LIN {X 0,Y 221.145,Z 638.431,A -85,B 0,C 180,E1 -21909.464,E2 -21909.464} C_VEL
LIN {X 0,Y 225.673,Z 625.218,A -85,B 0,C 180,E1 -21911.415,E2 -21911.415} C_VEL
LIN {X 0,Y 229.459,Z 612.073,A -85,B 0,C 180,E1 -21912.96,E2 -21912.96} C_VEL
LIN {X 0,Y 232.879,Z 597.827,A -85,B 0,C 180,E1 -21914.257,E2 -21914.257} C_VEL
LIN {X 0,Y 235.879,Z 582.403,A -85,B 0,C 180,E1 -21915.269,E2 -21915.269} C_VEL
LIN {X 0,Y 237.953,Z 566.942,A -85,B 0,C 180,E1 -21915.972,E2 -21915.972} C_VEL
LIN {X 0,Y 240.422,Z 531.68,A -85,B 0,C 180,E1 -21916.953,E2 -21916.953} C_VEL
LIN {X 0,Y 244.484,Z 467.241,A -85,B 0,C 180,E1 -21918.681,E2 -21918.681} C_VEL
LIN {X 0,Y 239.527,Z 455.727,A -85,B 0,C 180,E1 -21920.57,E2 -21920.57} C_VEL
LIN {X 0,Y 234.309,Z 445.003,A -85,B 0,C 180,E1 -21922.666,E2 -21922.666} C_VEL
LIN {X 0,Y 227.784,Z 433.109,A -85,B 0,C 180,E1 -21925.503,E2 -21925.503} C_VEL
LIN {X 0,Y 221.655,Z 423.149,A -85,B 0,C 180,E1 -21928.464,E2 -21928.464} C_VEL
LIN {X 0,Y 217.57,Z 417.19,A -85,B 0,C 180,E1 -21930.641,E2 -21930.641} C_VEL
LIN {X 0,Y 213.973,Z 412.042,A -85,B 0,C 180,E1 -21932.756,E2 -21932.756} C_VEL
LIN {X 0,Y 209.301,Z 405.782,A -85,B 0,C 180,E1 -21935.843,E2 -21935.843} C_VEL
LIN {X 0,Y 204.867,Z 400.056,A -85,B 0,C 180,E1 -21939.298,E2 -21939.298} C_VEL
LIN {X 0,Y 200.557,Z 394.827,A -85,B 0,C 180,E1 -21943.458,E2 -21943.458} C_VEL
LIN {X 0,Y 198.701,Z 391.203,A -85,B 0,C 180,E1 -21947.747,E2 -21947.747} C_VEL
LIN {X 0,Y 197.369,Z 389.174,A -85,B 0,C 180,E1 -21951.811,E2 -21951.811} C_VEL
LIN {X 0,Y 196.672,Z 386.877,A -85,B 0,C 180,E1 -21957.952,E2 -21957.952} C_VEL
LIN {X 0,Y 196.702,Z 386.437,A -85,B 0,C 180,E1 -21960,E2 -21960} C_VEL
LIN {X 0,Y 196.636,Z 386.629,A -85,B 0,C 180,E1 -21962.048,E2 -21962.048} C_VEL
LIN {X 0,Y 197.132,Z 388.567,A -85,B 0,C 180,E1 -21968.198,E2 -21968.198} C_VEL
LIN {X 0,Y 199.318,Z 391.66,A -85,B 0,C 180,E1 -21974.289,E2 -21974.289} C_VEL
LIN {X 0,Y 199.881,Z 392.9,A -85,B 0,C 180,E1 -21975.695,E2 -21975.695} C_VEL
LIN {X 0,Y 200.923,Z 394.996,A -85,B 0,C 180,E1 -21977.237,E2 -21977.237} C_VEL
LIN {X 0,Y 202.106,Z 398.063,A -85,B 0,C 180,E1 -21978.639,E2 -21978.639} C_VEL
LIN {X 0,Y 205.482,Z 407.511,A -85,B 0,C 180,E1 -21982.147,E2 -21982.147} C_VEL
LIN {X 0,Y 206.581,Z 409.464,A -85,B 0,C 180,E1 -21983.069,E2 -21983.069} C_VEL
LIN {X 0,Y 210.001,Z 413.782,A -85,B 0,C 180,E1 -21985.523,E2 -21985.523} C_VEL
LIN {X 0,Y 213.678,Z 418.756,A -85,B 0,C 180,E1 -21987.882,E2 -21987.882} C_VEL
LIN {X 0,Y 217.594,Z 424.126,A -85,B 0,C 180,E1 -21990.134,E2 -21990.134} C_VEL
LIN {X 0,Y 222.494,Z 431.302,A -85,B 0,C 180,E1 -21992.678,E2 -21992.678} C_VEL
LIN {X 0,Y 228.634,Z 440.96,A -85,B 0,C 180,E1 -21995.532,E2 -21995.532} C_VEL
LIN {X 0,Y 234.218,Z 450.7,A -85,B 0,C 180,E1 -21997.893,E2 -21997.893} C_VEL
LIN {X 0,Y 239.469,Z 465.456,A -85,B 0,C 180,E1 -22000.165,E2 -22000.165} C_VEL
LIN {X 0,Y 232.939,Z 563.19,A -85,B 0,C 180,E1 -22002.817,E2 -22002.817} C_VEL
LIN {X 0,Y 231.11,Z 578.287,A -85,B 0,C 180,E1 -22003.445,E2 -22003.445} C_VEL
LIN {X 0,Y 228.399,Z 593.01,A -85,B 0,C 180,E1 -22004.323,E2 -22004.323} C_VEL
LIN {X 0,Y 225.305,Z 606.361,A -85,B 0,C 180,E1 -22005.425,E2 -22005.425} C_VEL
LIN {X 0,Y 221.488,Z 620.138,A -85,B 0,C 180,E1 -22006.924,E2 -22006.924} C_VEL
LIN {X 0,Y 217.136,Z 633.278,A -85,B 0,C 180,E1 -22008.74,E2 -22008.74} C_VEL
LIN {X 0,Y 212.533,Z 645.127,A -85,B 0,C 180,E1 -22010.771,E2 -22010.771} C_VEL
LIN {X 0,Y 207.922,Z 656.085,A -85,B 0,C 180,E1 -22013.133,E2 -22013.133} C_VEL
LIN {X 0,Y 203.231,Z 666.179,A -85,B 0,C 180,E1 -22015.81,E2 -22015.81} C_VEL
LIN {X 0,Y 199.177,Z 674.689,A -85,B 0,C 180,E1 -22018.637,E2 -22018.637} C_VEL
LIN {X 0,Y 194.766,Z 683.074,A -85,B 0,C 180,E1 -22022.025,E2 -22022.025} C_VEL
LIN {X 0,Y 190.712,Z 690.93,A -85,B 0,C 180,E1 -22026.086,E2 -22026.086} C_VEL
LIN {X 0,Y 187.54,Z 697.179,A -85,B 0,C 180,E1 -22030.289,E2 -22030.289} C_VEL
LIN {X 0,Y 185.261,Z 701.999,A -85,B 0,C 180,E1 -22034.601,E2 -22034.601} C_VEL
LIN {X 0,Y 183.848,Z 705.52,A -85,B 0,C 180,E1 -22038.981,E2 -22038.981} C_VEL
LIN {X 0,Y 183.137,Z 707.835,A -85,B 0,C 180,E1 -22043.389,E2 -22043.389} C_VEL
LIN {X 0,Y 183.02,Z 708.996,A -85,B 0,C 180,E1 -22047.8,E2 -22047.8} C_VEL
LIN {X 0,Y 183.031,Z 709.146,A -85,B 0,C 180,E1 -22050,E2 -22050} C_VEL
LIN {X 0,Y 183.073,Z 708.547,A -85,B 0,C 180,E1 -22054.404,E2 -22054.404} C_VEL
LIN {X 0,Y 183.407,Z 706.799,A -85,B 0,C 180,E1 -22058.817,E2 -22058.817} C_VEL
LIN {X 0,Y 184.445,Z 703.868,A -85,B 0,C 180,E1 -22063.216,E2 -22063.216} C_VEL
LIN {X 0,Y 186.337,Z 699.686,A -85,B 0,C 180,E1 -22067.562,E2 -22067.562} C_VEL
LIN {X 0,Y 188.987,Z 694.152,A -85,B 0,C 180,E1 -22071.832,E2 -22071.832} C_VEL
LIN {X 0,Y 191.461,Z 689.781,A -85,B 0,C 180,E1 -22074.68,E2 -22074.68} C_VEL
LIN {X 0,Y 197.957,Z 686.616,A -85,B 0,C 180,E1 -22079.804,E2 -22079.804} C_VEL
LIN {X 0,Y 204.195,Z 683.167,A -85,B 0,C 180,E1 -22083.415,E2 -22083.415} C_VEL
LIN {X 0,Y 211.419,Z 678.76,A -85,B 0,C 180,E1 -22086.753,E2 -22086.753} C_VEL
LIN {X 0,Y 221.903,Z 671.855,A -85,B 0,C 180,E1 -22090.487,E2 -22090.487} C_VEL
LIN {X 0,Y 231.146,Z 665.173,A -85,B 0,C 180,E1 -22093.166,E2 -22093.166} C_VEL
LIN {X 0,Y 242.53,Z 656.247,A -85,B 0,C 180,E1 -22095.824,E2 -22095.824} C_VEL
LIN {X 0,Y 246.76,Z 652.737,A -85,B 0,C 180,E1 -22096.694,E2 -22096.694} C_VEL
LIN {X 0,Y 248.311,Z 651.353,A -85,B 0,C 180,E1 -22097.213,E2 -22097.213} C_VEL
LIN {X 0,Y 238.076,Z 658.959,A -85,B 0,C 180,E1 -22099.501,E2 -22099.501} C_VEL
LIN {X 0,Y 228.584,Z 665.287,A -85,B 0,C 180,E1 -22102.054,E2 -22102.054} C_VEL
LIN {X 0,Y 219.85,Z 670.441,A -85,B 0,C 180,E1 -22104.872,E2 -22104.872} C_VEL
LIN {X 0,Y 211.838,Z 674.517,A -85,B 0,C 180,E1 -22107.939,E2 -22107.939} C_VEL
LIN {X 0,Y 204.688,Z 677.495,A -85,B 0,C 180,E1 -22111.27,E2 -22111.27} C_VEL
LIN {X 0,Y 198.621,Z 679.336,A -85,B 0,C 180,E1 -22114.874,E2 -22114.874} C_VEL
LIN {X 0,Y 193.513,Z 680.122,A -85,B 0,C 180,E1 -22118.705,E2 -22118.705} C_VEL
LIN {X 0,Y 189.625,Z 679.823,A -85,B 0,C 180,E1 -22122.753,E2 -22122.753} C_VEL
LIN {X 0,Y 186.665,Z 678.421,A -85,B 0,C 180,E1 -22126.944,E2 -22126.944} C_VEL
LIN {X 0,Y 184.683,Z 675.852,A -85,B 0,C 180,E1 -22131.245,E2 -22131.245} C_VEL
LIN {X 0,Y 183.798,Z 672.043,A -85,B 0,C 180,E1 -22135.614,E2 -22135.614} C_VEL
LIN {X 0,Y 183.535,Z 668.25,A -85,B 0,C 180,E1 -22138.903,E2 -22138.903} C_VEL
LIN {X 0,Y 183.475,Z 663.633,A -85,B 0,C 180,E1 -22142.195,E2 -22142.195} C_VEL
LIN {X 0,Y 183.761,Z 655.877,A -85,B 0,C 180,E1 -22146.589,E2 -22146.589} C_VEL
LIN {X 0,Y 184.363,Z 647.395,A -85,B 0,C 180,E1 -22150.432,E2 -22150.432} C_VEL
LIN {X 0,Y 185.232,Z 638.646,A -85,B 0,C 180,E1 -22153.718,E2 -22153.718} C_VEL
LIN {X 0,Y 186.582,Z 628.253,A -85,B 0,C 180,E1 -22156.973,E2 -22156.973} C_VEL
LIN {X 0,Y 188.232,Z 616.073,A -85,B 0,C 180,E1 -22160.138,E2 -22160.138} C_VEL
LIN {X 0,Y 190.004,Z 603.327,A -85,B 0,C 180,E1 -22162.853,E2 -22162.853} C_VEL
LIN {X 0,Y 191.936,Z 589.886,A -85,B 0,C 180,E1 -22165.193,E2 -22165.193} C_VEL
LIN {X 0,Y 193.983,Z 574.43,A -85,B 0,C 180,E1 -22167.366,E2 -22167.366} C_VEL
LIN {X 0,Y 194.89,Z 567.266,A -85,B 0,C 180,E1 -22168.396,E2 -22168.396} C_VEL
LIN {X 0,Y 195.611,Z 564.799,A -85,B 0,C 180,E1 -22169.015,E2 -22169.015} C_VEL
LIN {X 0,Y 197.306,Z 562.863,A -85,B 0,C 180,E1 -22169.839,E2 -22169.839} C_VEL
LIN {X 0,Y 199.619,Z 558.803,A -85,B 0,C 180,E1 -22170.624,E2 -22170.624} C_VEL
LIN {X 0,Y 202.727,Z 550.321,A -85,B 0,C 180,E1 -22171.506,E2 -22171.506} C_VEL
LIN {X 0,Y 207.709,Z 533.515,A -85,B 0,C 180,E1 -22172.634,E2 -22172.634} C_VEL
LIN {X 0,Y 209.994,Z 530.321,A -85,B 0,C 180,E1 -22173.397,E2 -22173.397} C_VEL
LIN {X 0,Y 212.304,Z 525.327,A -85,B 0,C 180,E1 -22174.034,E2 -22174.034} C_VEL
LIN {X 0,Y 216.015,Z 514.502,A -85,B 0,C 180,E1 -22174.848,E2 -22174.848} C_VEL
LIN {X 0,Y 221.035,Z 497.363,A -85,B 0,C 180,E1 -22175.746,E2 -22175.746} C_VEL
LIN {X 0,Y 223.977,Z 492.781,A -85,B 0,C 180,E1 -22176.534,E2 -22176.534} C_VEL
LIN {X 0,Y 227.199,Z 485.435,A -85,B 0,C 180,E1 -22177.239,E2 -22177.239} C_VEL
LIN {X 0,Y 230.92,Z 474.319,A -85,B 0,C 180,E1 -22177.885,E2 -22177.885} C_VEL
LIN {X 0,Y 234.212,Z 463.118,A -85,B 0,C 180,E1 -22178.366,E2 -22178.366} C_VEL
LIN {X 0,Y 235.788,Z 461.138,A -85,B 0,C 180,E1 -22178.751,E2 -22178.751} C_VEL
LIN {X 0,Y 238.047,Z 465.902,A -85,B 0,C 180,E1 -22179.642,E2 -22179.642} C_VEL
LIN {X 0,Y 239.544,Z 469.549,A -85,B 0,C 180,E1 -22180.237,E2 -22180.237} C_VEL
LIN {X 0,Y 234.668,Z 543.882,A -85,B 0,C 180,E1 -22182.243,E2 -22182.243} C_VEL
LIN {X 0,Y 232.919,Z 566.712,A -85,B 0,C 180,E1 -22182.89,E2 -22182.89} C_VEL
LIN {X 0,Y 230.795,Z 582.245,A -85,B 0,C 180,E1 -22183.6,E2 -22183.6} C_VEL
LIN {X 0,Y 227.711,Z 597.718,A -85,B 0,C 180,E1 -22184.619,E2 -22184.619} C_VEL
LIN {X 0,Y 224.425,Z 611.093,A -85,B 0,C 180,E1 -22185.831,E2 -22185.831} C_VEL
LIN {X 0,Y 220.636,Z 624.081,A -85,B 0,C 180,E1 -22187.36,E2 -22187.36} C_VEL
LIN {X 0,Y 215.819,Z 637.746,A -85,B 0,C 180,E1 -22189.361,E2 -22189.361} C_VEL
LIN {X 0,Y 210.958,Z 649.959,A -85,B 0,C 180,E1 -22191.648,E2 -22191.648} C_VEL
LIN {X 0,Y 205.603,Z 661.938,A -85,B 0,C 180,E1 -22194.472,E2 -22194.472} C_VEL
LIN {X 0,Y 200.757,Z 672.218,A -85,B 0,C 180,E1 -22197.57,E2 -22197.57} C_VEL
LIN {X 0,Y 196.656,Z 680.261,A -85,B 0,C 180,E1 -22200.568,E2 -22200.568} C_VEL
LIN {X 0,Y 192.717,Z 687.801,A -85,B 0,C 180,E1 -22204.048,E2 -22204.048} C_VEL
LIN {X 0,Y 189.086,Z 694.833,A -85,B 0,C 180,E1 -22208.18,E2 -22208.18} C_VEL
LIN {X 0,Y 186.404,Z 700.363,A -85,B 0,C 180,E1 -22212.445,E2 -22212.445} C_VEL
LIN {X 0,Y 184.461,Z 704.547,A -85,B 0,C 180,E1 -22216.785,E2 -22216.785} C_VEL
LIN {X 0,Y 183.41,Z 707.485,A -85,B 0,C 180,E1 -22221.183,E2 -22221.183} C_VEL
LIN {X 0,Y 183.015,Z 709.245,A -85,B 0,C 180,E1 -22225.595,E2 -22225.595} C_VEL
LIN {X 0,Y 183.028,Z 709.852,A -85,B 0,C 180,E1 -22230,E2 -22230} C_VEL
LIN {X 0,Y 183.015,Z 709.275,A -85,B 0,C 180,E1 -22234.405,E2 -22234.405} C_VEL
LIN {X 0,Y 183.409,Z 707.556,A -85,B 0,C 180,E1 -22238.816,E2 -22238.816} C_VEL
LIN {X 0,Y 184.449,Z 704.665,A -85,B 0,C 180,E1 -22243.215,E2 -22243.215} C_VEL
LIN {X 0,Y 186.36,Z 700.533,A -85,B 0,C 180,E1 -22247.559,E2 -22247.559} C_VEL
LIN {X 0,Y 188.988,Z 695.048,A -85,B 0,C 180,E1 -22251.831,E2 -22251.831} C_VEL
LIN {X 0,Y 192.642,Z 688.063,A -85,B 0,C 180,E1 -22255.962,E2 -22255.962} C_VEL
LIN {X 0,Y 196.578,Z 680.583,A -85,B 0,C 180,E1 -22259.445,E2 -22259.445} C_VEL
LIN {X 0,Y 200.549,Z 672.82,A -85,B 0,C 180,E1 -22262.359,E2 -22262.359} C_VEL
LIN {X 0,Y 204.713,Z 663.972,A -85,B 0,C 180,E1 -22265.102,E2 -22265.102} C_VEL
LIN {X 0,Y 209.575,Z 653.397,A -85,B 0,C 180,E1 -22267.734,E2 -22267.734} C_VEL
LIN {X 0,Y 214.332,Z 641.871,A -85,B 0,C 180,E1 -22270.054,E2 -22270.054} C_VEL
LIN {X 0,Y 218.996,Z 629.303,A -85,B 0,C 180,E1 -22272.06,E2 -22272.06} C_VEL
LIN {X 0,Y 223.324,Z 615.487,A -85,B 0,C 180,E1 -22273.815,E2 -22273.815} C_VEL
LIN {X 0,Y 227.053,Z 601.067,A -85,B 0,C 180,E1 -22275.234,E2 -22275.234} C_VEL
LIN {X 0,Y 230.223,Z 586.022,A -85,B 0,C 180,E1 -22276.311,E2 -22276.311} C_VEL
LIN {X 0,Y 232.53,Z 571.213,A -85,B 0,C 180,E1 -22277.053,E2 -22277.053} C_VEL
LIN {X 0,Y 234.057,Z 554.756,A -85,B 0,C 180,E1 -22277.601,E2 -22277.601} C_VEL
LIN {X 0,Y 239.721,Z 469.822,A -85,B 0,C 180,E1 -22279.869,E2 -22279.869} C_VEL
LIN {X 0,Y 235.05,Z 458.909,A -85,B 0,C 180,E1 -22281.755,E2 -22281.755} C_VEL
LIN {X 0,Y 230.72,Z 449.849,A -85,B 0,C 180,E1 -22283.595,E2 -22283.595} C_VEL
LIN {X 0,Y 224.812,Z 438.744,A -85,B 0,C 180,E1 -22286.296,E2 -22286.296} C_VEL
LIN {X 0,Y 219.094,Z 429.197,A -85,B 0,C 180,E1 -22289.187,E2 -22289.187} C_VEL
LIN {X 0,Y 215.01,Z 423.058,A -85,B 0,C 180,E1 -22291.467,E2 -22291.467} C_VEL
LIN {X 0,Y 211.775,Z 418.254,A -85,B 0,C 180,E1 -22293.463,E2 -22293.463} C_VEL
LIN {X 0,Y 207.224,Z 411.967,A -85,B 0,C 180,E1 -22296.615,E2 -22296.615} C_VEL
LIN {X 0,Y 203.203,Z 406.629,A -85,B 0,C 180,E1 -22299.897,E2 -22299.897} C_VEL
LIN {X 0,Y 199.028,Z 401.431,A -85,B 0,C 180,E1 -22304.107,E2 -22304.107} C_VEL
LIN {X 0,Y 195.577,Z 397.2,A -85,B 0,C 180,E1 -22308.863,E2 -22308.863} C_VEL
LIN {X 0,Y 193.057,Z 394.152,A -85,B 0,C 180,E1 -22314.778,E2 -22314.778} C_VEL
LIN {X 0,Y 192.936,Z 392.985,A -85,B 0,C 180,E1 -22317.912,E2 -22317.912} C_VEL
LIN {X 0,Y 193.023,Z 392.513,A -85,B 0,C 180,E1 -22320,E2 -22320} C_VEL
LIN {X 0,Y 192.98,Z 392.732,A -85,B 0,C 180,E1 -22322.087,E2 -22322.087} C_VEL
LIN {X 0,Y 193.62,Z 394.522,A -85,B 0,C 180,E1 -22327.299,E2 -22327.299} C_VEL
LIN {X 0,Y 197.673,Z 398.839,A -85,B 0,C 180,E1 -22334.411,E2 -22334.411} C_VEL
LIN {X 0,Y 202.371,Z 404.31,A -85,B 0,C 180,E1 -22339.527,E2 -22339.527} C_VEL
LIN {X 0,Y 206.581,Z 409.464,A -85,B 0,C 180,E1 -22343.069,E2 -22343.069} C_VEL
LIN {X 0,Y 208.227,Z 412.598,A -85,B 0,C 180,E1 -22344.376,E2 -22344.376} C_VEL
LIN {X 0,Y 213.629,Z 427.51,A -85,B 0,C 180,E1 -22348.471,E2 -22348.471} C_VEL
LIN {X 0,Y 214.927,Z 429.826,A -85,B 0,C 180,E1 -22349.263,E2 -22349.263} C_VEL
LIN {X 0,Y 219.451,Z 436.637,A -85,B 0,C 180,E1 -22351.737,E2 -22351.737} C_VEL
LIN {X 0,Y 225.346,Z 446.156,A -85,B 0,C 180,E1 -22354.625,E2 -22354.625} C_VEL
LIN {X 0,Y 230.661,Z 455.683,A -85,B 0,C 180,E1 -22356.99,E2 -22356.99} C_VEL
LIN {X 0,Y 234.817,Z 467.821,A -85,B 0,C 180,E1 -22358.907,E2 -22358.907} C_VEL
LIN {X 0,Y 228.174,Z 563.309,A -85,B 0,C 180,E1 -22361.509,E2 -22361.509} C_VEL
LIN {X 0,Y 226.298,Z 578.362,A -85,B 0,C 180,E1 -22362.143,E2 -22362.143} C_VEL
LIN {X 0,Y 223.509,Z 593.064,A -85,B 0,C 180,E1 -22363.024,E2 -22363.024} C_VEL
LIN {X 0,Y 220.303,Z 606.404,A -85,B 0,C 180,E1 -22364.129,E2 -22364.129} C_VEL
LIN {X 0,Y 216.479,Z 619.733,A -85,B 0,C 180,E1 -22365.58,E2 -22365.58} C_VEL
LIN {X 0,Y 211.849,Z 633.307,A -85,B 0,C 180,E1 -22367.474,E2 -22367.474} C_VEL
LIN {X 0,Y 207.08,Z 645.152,A -85,B 0,C 180,E1 -22369.528,E2 -22369.528} C_VEL
LIN {X 0,Y 202.257,Z 656.108,A -85,B 0,C 180,E1 -22371.919,E2 -22371.919} C_VEL
LIN {X 0,Y 197.372,Z 666.2,A -85,B 0,C 180,E1 -22374.646,E2 -22374.646} C_VEL
LIN {X 0,Y 194.301,Z 672.289,A -85,B 0,C 180,E1 -22376.646,E2 -22376.646} C_VEL
LIN {X 0,Y 189.721,Z 680.876,A -85,B 0,C 180,E1 -22379.994,E2 -22379.994} C_VEL
LIN {X 0,Y 185.167,Z 689.149,A -85,B 0,C 180,E1 -22384.121,E2 -22384.121} C_VEL
LIN {X 0,Y 181.661,Z 695.501,A -85,B 0,C 180,E1 -22388.202,E2 -22388.202} C_VEL
LIN {X 0,Y 178.942,Z 700.957,A -85,B 0,C 180,E1 -22392.869,E2 -22392.869} C_VEL
LIN {X 0,Y 177.481,Z 703.93,A -85,B 0,C 180,E1 -22396.256,E2 -22396.256} C_VEL
LIN {X 0,Y 176.353,Z 706.839,A -85,B 0,C 180,E1 -22400.828,E2 -22400.828} C_VEL
LIN {X 0,Y 175.969,Z 708.572,A -85,B 0,C 180,E1 -22405.419,E2 -22405.419} C_VEL
LIN {X 0,Y 175.946,Z 709.16,A -85,B 0,C 180,E1 -22410,E2 -22410} C_VEL
LIN {X 0,Y 175.97,Z 708.561,A -85,B 0,C 180,E1 -22414.582,E2 -22414.582} C_VEL
LIN {X 0,Y 176.353,Z 706.812,A -85,B 0,C 180,E1 -22419.173,E2 -22419.173} C_VEL
LIN {X 0,Y 177.483,Z 703.881,A -85,B 0,C 180,E1 -22423.745,E2 -22423.745} C_VEL
LIN {X 0,Y 179.514,Z 699.7,A -85,B 0,C 180,E1 -22428.253,E2 -22428.253} C_VEL
LIN {X 0,Y 182.354,Z 694.166,A -85,B 0,C 180,E1 -22432.669,E2 -22432.669} C_VEL
LIN {X 0,Y 184.976,Z 689.731,A -85,B 0,C 180,E1 -22435.607,E2 -22435.607} C_VEL
LIN {X 0,Y 191.816,Z 686.999,A -85,B 0,C 180,E1 -22440.861,E2 -22440.861} C_VEL
LIN {X 0,Y 198.348,Z 683.928,A -85,B 0,C 180,E1 -22444.536,E2 -22444.536} C_VEL
LIN {X 0,Y 205.866,Z 679.965,A -85,B 0,C 180,E1 -22447.916,E2 -22447.916} C_VEL
LIN {X 0,Y 216.709,Z 673.66,A -85,B 0,C 180,E1 -22451.669,E2 -22451.669} C_VEL
LIN {X 0,Y 228.77,Z 665.813,A -85,B 0,C 180,E1 -22454.958,E2 -22454.958} C_VEL
LIN {X 0,Y 237.539,Z 659.537,A -85,B 0,C 180,E1 -22456.909,E2 -22456.909} C_VEL
LIN {X 0,Y 238.3,Z 658.944,A -85,B 0,C 180,E1 -22457.288,E2 -22457.288} C_VEL
LIN {X 0,Y 228.177,Z 665.279,A -85,B 0,C 180,E1 -22459.698,E2 -22459.698} C_VEL
LIN {X 0,Y 218.763,Z 670.502,A -85,B 0,C 180,E1 -22462.382,E2 -22462.382} C_VEL
LIN {X 0,Y 210.096,Z 674.614,A -85,B 0,C 180,E1 -22465.343,E2 -22465.343} C_VEL
LIN {X 0,Y 202.137,Z 677.686,A -85,B 0,C 180,E1 -22468.566,E2 -22468.566} C_VEL
LIN {X 0,Y 195.325,Z 679.663,A -85,B 0,C 180,E1 -22472.112,E2 -22472.112} C_VEL
LIN {X 0,Y 189.461,Z 680.637,A -85,B 0,C 180,E1 -22475.918,E2 -22475.918} C_VEL
LIN {X 0,Y 184.785,Z 680.556,A -85,B 0,C 180,E1 -22479.983,E2 -22479.983} C_VEL
LIN {X 0,Y 181.163,Z 679.359,A -85,B 0,C 180,E1 -22484.243,E2 -22484.243} C_VEL
LIN {X 0,Y 178.611,Z 677.044,A -85,B 0,C 180,E1 -22488.654,E2 -22488.654} C_VEL
LIN {X 0,Y 177.05,Z 673.543,A -85,B 0,C 180,E1 -22493.161,E2 -22493.161} C_VEL
LIN {X 0,Y 176.576,Z 668.761,A -85,B 0,C 180,E1 -22497.719,E2 -22497.719} C_VEL
LIN {X 0,Y 176.452,Z 664.212,A -85,B 0,C 180,E1 -22501.141,E2 -22501.141} C_VEL
LIN {X 0,Y 176.59,Z 657.403,A -85,B 0,C 180,E1 -22505.267,E2 -22505.267} C_VEL
LIN {X 0,Y 177.114,Z 649.531,A -85,B 0,C 180,E1 -22509.133,E2 -22509.133} C_VEL
LIN {X 0,Y 178.03,Z 639.591,A -85,B 0,C 180,E1 -22513.12,E2 -22513.12} C_VEL
LIN {X 0,Y 179.321,Z 629.357,A -85,B 0,C 180,E1 -22516.508,E2 -22516.508} C_VEL
LIN {X 0,Y 180.953,Z 617.112,A -85,B 0,C 180,E1 -22519.867,E2 -22519.867} C_VEL
LIN {X 0,Y 182.858,Z 603.514,A -85,B 0,C 180,E1 -22522.902,E2 -22522.902} C_VEL
LIN {X 0,Y 185.215,Z 587.713,A -85,B 0,C 180,E1 -22525.873,E2 -22525.873} C_VEL
LIN {X 0,Y 185.81,Z 585.76,A -85,B 0,C 180,E1 -22526.538,E2 -22526.538} C_VEL
LIN {X 0,Y 186.309,Z 585.526,A -85,B 0,C 180,E1 -22526.915,E2 -22526.915} C_VEL
LIN {X 0,Y 188.814,Z 583.488,A -85,B 0,C 180,E1 -22528.03,E2 -22528.03} C_VEL
LIN {X 0,Y 191.85,Z 579.114,A -85,B 0,C 180,E1 -22528.985,E2 -22528.985} C_VEL
LIN {X 0,Y 196.432,Z 570.642,A -85,B 0,C 180,E1 -22530.201,E2 -22530.201} C_VEL
LIN {X 0,Y 198.964,Z 568.102,A -85,B 0,C 180,E1 -22531.141,E2 -22531.141} C_VEL
LIN {X 0,Y 201.887,Z 563.31,A -85,B 0,C 180,E1 -22532.06,E2 -22532.06} C_VEL
LIN {X 0,Y 205.229,Z 555.197,A -85,B 0,C 180,E1 -22532.932,E2 -22532.932} C_VEL
LIN {X 0,Y 209.055,Z 542.703,A -85,B 0,C 180,E1 -22533.763,E2 -22533.763} C_VEL
LIN {X 0,Y 210.533,Z 537.912,A -85,B 0,C 180,E1 -22534.073,E2 -22534.073} C_VEL
LIN {X 0,Y 213.531,Z 533.131,A -85,B 0,C 180,E1 -22534.967,E2 -22534.967} C_VEL
LIN {X 0,Y 216.361,Z 526.461,A -85,B 0,C 180,E1 -22535.651,E2 -22535.651} C_VEL
LIN {X 0,Y 220.395,Z 514.599,A -85,B 0,C 180,E1 -22536.45,E2 -22536.45} C_VEL
LIN {X 0,Y 224.382,Z 501.19,A -85,B 0,C 180,E1 -22537.111,E2 -22537.111} C_VEL
LIN {X 0,Y 227.51,Z 496.004,A -85,B 0,C 180,E1 -22537.876,E2 -22537.876} C_VEL
LIN {X 0,Y 230.897,Z 488.304,A -85,B 0,C 180,E1 -22538.566,E2 -22538.566} C_VEL
LIN {X 0,Y 234.446,Z 478.064,A -85,B 0,C 180,E1 -22539.153,E2 -22539.153} C_VEL
LIN {X 0,Y 228.554,Z 562.464,A -85,B 0,C 180,E1 -22541.45,E2 -22541.45} C_VEL
LIN {X 0,Y 226.647,Z 577.85,A -85,B 0,C 180,E1 -22542.074,E2 -22542.074} C_VEL
LIN {X 0,Y 223.909,Z 592.734,A -85,B 0,C 180,E1 -22542.968,E2 -22542.968} C_VEL
LIN {X 0,Y 220.934,Z 605.251,A -85,B 0,C 180,E1 -22543.969,E2 -22543.969} C_VEL
LIN {X 0,Y 216.836,Z 619.529,A -85,B 0,C 180,E1 -22545.484,E2 -22545.484} C_VEL
LIN {X 0,Y 212.439,Z 632.65,A -85,B 0,C 180,E1 -22547.297,E2 -22547.297} C_VEL
LIN {X 0,Y 207.644,Z 644.67,A -85,B 0,C 180,E1 -22549.342,E2 -22549.342} C_VEL
LIN {X 0,Y 202.345,Z 656.668,A -85,B 0,C 180,E1 -22551.938,E2 -22551.938} C_VEL
LIN {X 0,Y 197.463,Z 666.742,A -85,B 0,C 180,E1 -22554.664,E2 -22554.664} C_VEL
LIN {X 0,Y 192.548,Z 676.581,A -85,B 0,C 180,E1 -22558.045,E2 -22558.045} C_VEL
LIN {X 0,Y 187.997,Z 684.746,A -85,B 0,C 180,E1 -22561.533,E2 -22561.533} C_VEL
LIN {X 0,Y 184.242,Z 691.503,A -85,B 0,C 180,E1 -22565.19,E2 -22565.19} C_VEL
LIN {X 0,Y 180.904,Z 697.76,A -85,B 0,C 180,E1 -22569.534,E2 -22569.534} C_VEL
LIN {X 0,Y 178.431,Z 702.602,A -85,B 0,C 180,E1 -22573.995,E2 -22573.995} C_VEL
LIN {X 0,Y 176.861,Z 706.154,A -85,B 0,C 180,E1 -22578.54,E2 -22578.54} C_VEL
LIN {X 0,Y 176.074,Z 708.495,A -85,B 0,C 180,E1 -22583.122,E2 -22583.122} C_VEL
LIN {X 0,Y 175.888,Z 709.682,A -85,B 0,C 180,E1 -22587.71,E2 -22587.71} C_VEL
LIN {X 0,Y 175.937,Z 709.839,A -85,B 0,C 180,E1 -22590,E2 -22590} C_VEL
LIN {X 0,Y 175.936,Z 709.261,A -85,B 0,C 180,E1 -22594.582,E2 -22594.582} C_VEL
LIN {X 0,Y 176.355,Z 707.542,A -85,B 0,C 180,E1 -22599.172,E2 -22599.172} C_VEL
LIN {X 0,Y 177.488,Z 704.65,A -85,B 0,C 180,E1 -22603.744,E2 -22603.744} C_VEL
LIN {X 0,Y 179.536,Z 700.517,A -85,B 0,C 180,E1 -22608.25,E2 -22608.25} C_VEL
LIN {X 0,Y 182.356,Z 695.031,A -85,B 0,C 180,E1 -22612.668,E2 -22612.668} C_VEL
LIN {X 0,Y 186.24,Z 688.045,A -85,B 0,C 180,E1 -22616.926,E2 -22616.926} C_VEL
LIN {X 0,Y 190.404,Z 680.564,A -85,B 0,C 180,E1 -22620.499,E2 -22620.499} C_VEL
LIN {X 0,Y 194.913,Z 671.914,A -85,B 0,C 180,E1 -22623.821,E2 -22623.821} C_VEL
LIN {X 0,Y 199.73,Z 662.342,A -85,B 0,C 180,E1 -22626.74,E2 -22626.74} C_VEL
LIN {X 0,Y 205.273,Z 650.481,A -85,B 0,C 180,E1 -22629.618,E2 -22629.618} C_VEL
LIN {X 0,Y 210.356,Z 638.375,A -85,B 0,C 180,E1 -22631.928,E2 -22631.928} C_VEL
LIN {X 0,Y 215.342,Z 624.759,A -85,B 0,C 180,E1 -22633.972,E2 -22633.972} C_VEL
LIN {X 0,Y 219.265,Z 611.997,A -85,B 0,C 180,E1 -22635.493,E2 -22635.493} C_VEL
LIN {X 0,Y 222.925,Z 597.732,A -85,B 0,C 180,E1 -22636.806,E2 -22636.806} C_VEL
LIN {X 0,Y 226.123,Z 582.27,A -85,B 0,C 180,E1 -22637.823,E2 -22637.823} C_VEL
LIN {X 0,Y 228.314,Z 566.729,A -85,B 0,C 180,E1 -22638.534,E2 -22638.534} C_VEL
LIN {X 0,Y 231.309,Z 526.621,A -85,B 0,C 180,E1 -22639.651,E2 -22639.651} C_VEL
LIN {X 0,Y 234.946,Z 472.122,A -85,B 0,C 180,E1 -22641.153,E2 -22641.153} C_VEL
LIN {X 0,Y 230.11,Z 460.813,A -85,B 0,C 180,E1 -22643.238,E2 -22643.238} C_VEL
LIN {X 0,Y 225.358,Z 451.002,A -85,B 0,C 180,E1 -22645.412,E2 -22645.412} C_VEL
LIN {X 0,Y 219.661,Z 440.473,A -85,B 0,C 180,E1 -22648.25,E2 -22648.25} C_VEL
LIN {X 0,Y 214.757,Z 432.384,A -85,B 0,C 180,E1 -22650.958,E2 -22650.958} C_VEL
LIN {X 0,Y 212.47,Z 428.895,A -85,B 0,C 180,E1 -22652.327,E2 -22652.327} C_VEL
LIN {X 0,Y 209.64,Z 424.526,A -85,B 0,C 180,E1 -22654.163,E2 -22654.163} C_VEL
LIN {X 0,Y 205.404,Z 418.484,A -85,B 0,C 180,E1 -22657.228,E2 -22657.228} C_VEL
LIN {X 0,Y 201.546,Z 413.185,A -85,B 0,C 180,E1 -22660.522,E2 -22660.522} C_VEL
LIN {X 0,Y 197.548,Z 408.021,A -85,B 0,C 180,E1 -22664.764,E2 -22664.764} C_VEL
LIN {X 0,Y 194.415,Z 404.041,A -85,B 0,C 180,E1 -22669.323,E2 -22669.323} C_VEL
LIN {X 0,Y 192.079,Z 401.141,A -85,B 0,C 180,E1 -22675.015,E2 -22675.015} C_VEL
LIN {X 0,Y 191.511,Z 399.468,A -85,B 0,C 180,E1 -22680,E2 -22680} C_VEL
LIN {X 0,Y 191.777,Z 400.241,A -85,B 0,C 180,E1 -22683.677,E2 -22683.677} C_VEL
LIN {X 0,Y 193.158,Z 402.175,A -85,B 0,C 180,E1 -22688.368,E2 -22688.368} C_VEL
LIN {X 0,Y 196.61,Z 405.877,A -85,B 0,C 180,E1 -22694.213,E2 -22694.213} C_VEL
LIN {X 0,Y 200.801,Z 410.892,A -85,B 0,C 180,E1 -22698.939,E2 -22698.939} C_VEL
LIN {X 0,Y 204.925,Z 416.202,A -85,B 0,C 180,E1 -22702.562,E2 -22702.562} C_VEL
LIN {X 0,Y 208.148,Z 420.422,A -85,B 0,C 180,E1 -22704.964,E2 -22704.964} C_VEL
LIN {X 0,Y 211.565,Z 425.143,A -85,B 0,C 180,E1 -22707.243,E2 -22707.243} C_VEL
LIN {X 0,Y 214.927,Z 429.826,A -85,B 0,C 180,E1 -22709.263,E2 -22709.263} C_VEL
LIN {X 0,Y 216.797,Z 433.523,A -85,B 0,C 180,E1 -22710.377,E2 -22710.377} C_VEL
LIN {X 0,Y 219.222,Z 441.133,A -85,B 0,C 180,E1 -22711.914,E2 -22711.914} C_VEL
LIN {X 0,Y 222.11,Z 450.706,A -85,B 0,C 180,E1 -22713.651,E2 -22713.651} C_VEL
LIN {X 0,Y 223.361,Z 453.565,A -85,B 0,C 180,E1 -22714.294,E2 -22714.294} C_VEL
LIN {X 0,Y 227.072,Z 460.526,A -85,B 0,C 180,E1 -22716.019,E2 -22716.019} C_VEL
LIN {X 0,Y 230.26,Z 470.048,A -85,B 0,C 180,E1 -22717.583,E2 -22717.583} C_VEL
LIN {X 0,Y 223.548,Z 563.423,A -85,B 0,C 180,E1 -22720.151,E2 -22720.151} C_VEL
LIN {X 0,Y 221.604,Z 578.433,A -85,B 0,C 180,E1 -22720.784,E2 -22720.784} C_VEL
LIN {X 0,Y 218.741,Z 593.116,A -85,B 0,C 180,E1 -22721.668,E2 -22721.668} C_VEL
LIN {X 0,Y 215.414,Z 606.446,A -85,B 0,C 180,E1 -22722.771,E2 -22722.771} C_VEL
LIN {X 0,Y 211.205,Z 620.54,A -85,B 0,C 180,E1 -22724.33,E2 -22724.33} C_VEL
LIN {X 0,Y 206.163,Z 634.615,A -85,B 0,C 180,E1 -22726.345,E2 -22726.345} C_VEL
LIN {X 0,Y 200.76,Z 647.295,A -85,B 0,C 180,E1 -22728.643,E2 -22728.643} C_VEL
LIN {X 0,Y 195.816,Z 657.897,A -85,B 0,C 180,E1 -22731.091,E2 -22731.091} C_VEL
LIN {X 0,Y 190.762,Z 667.703,A -85,B 0,C 180,E1 -22733.881,E2 -22733.881} C_VEL
LIN {X 0,Y 187.1,Z 674.729,A -85,B 0,C 180,E1 -22736.355,E2 -22736.355} C_VEL
LIN {X 0,Y 182.246,Z 683.11,A -85,B 0,C 180,E1 -22739.913,E2 -22739.913} C_VEL
LIN {X 0,Y 177.713,Z 690.964,A -85,B 0,C 180,E1 -22744.214,E2 -22744.214} C_VEL
LIN {X 0,Y 174.131,Z 697.211,A -85,B 0,C 180,E1 -22748.701,E2 -22748.701} C_VEL
LIN {X 0,Y 171.549,Z 702.029,A -85,B 0,C 180,E1 -22753.335,E2 -22753.335} C_VEL
LIN {X 0,Y 169.859,Z 705.549,A -85,B 0,C 180,E1 -22758.061,E2 -22758.061} C_VEL
LIN {X 0,Y 168.998,Z 707.864,A -85,B 0,C 180,E1 -22762.833,E2 -22762.833} C_VEL
LIN {X 0,Y 168.837,Z 709.024,A -85,B 0,C 180,E1 -22767.615,E2 -22767.615} C_VEL
LIN {X 0,Y 168.849,Z 709.174,A -85,B 0,C 180,E1 -22770,E2 -22770} C_VEL
LIN {X 0,Y 168.873,Z 708.575,A -85,B 0,C 180,E1 -22774.775,E2 -22774.775} C_VEL
LIN {X 0,Y 169.321,Z 706.826,A -85,B 0,C 180,E1 -22779.557,E2 -22779.557} C_VEL
LIN {X 0,Y 170.542,Z 703.895,A -85,B 0,C 180,E1 -22784.316,E2 -22784.316} C_VEL
LIN {X 0,Y 172.709,Z 699.713,A -85,B 0,C 180,E1 -22788.999,E2 -22788.999} C_VEL
LIN {X 0,Y 175.764,Z 694.18,A -85,B 0,C 180,E1 -22793.569,E2 -22793.569} C_VEL
LIN {X 0,Y 178.578,Z 689.605,A -85,B 0,C 180,E1 -22796.594,E2 -22796.594} C_VEL
LIN {X 0,Y 185.745,Z 687.329,A -85,B 0,C 180,E1 -22801.987,E2 -22801.987} C_VEL
LIN {X 0,Y 196.326,Z 682.925,A -85,B 0,C 180,E1 -22807.486,E2 -22807.486} C_VEL
LIN {X 0,Y 204.735,Z 678.937,A -85,B 0,C 180,E1 -22810.709,E2 -22810.709} C_VEL
LIN {X 0,Y 216.432,Z 672.634,A -85,B 0,C 180,E1 -22814.279,E2 -22814.279} C_VEL
LIN {X 0,Y 225.588,Z 667.134,A -85,B 0,C 180,E1 -22816.546,E2 -22816.546} C_VEL
LIN {X 0,Y 228.273,Z 665.438,A -85,B 0,C 180,E1 -22817.365,E2 -22817.365} C_VEL
LIN {X 0,Y 215.805,Z 671.759,A -85,B 0,C 180,E1 -22820.577,E2 -22820.577} C_VEL
LIN {X 0,Y 204.49,Z 676.466,A -85,B 0,C 180,E1 -22824.249,E2 -22824.249} C_VEL
LIN {X 0,Y 196.249,Z 679.119,A -85,B 0,C 180,E1 -22827.509,E2 -22827.509} C_VEL
LIN {X 0,Y 189.165,Z 680.73,A -85,B 0,C 180,E1 -22831.12,E2 -22831.12} C_VEL
LIN {X 0,Y 183.043,Z 681.303,A -85,B 0,C 180,E1 -22835.017,E2 -22835.017} C_VEL
LIN {X 0,Y 178.125,Z 680.829,A -85,B 0,C 180,E1 -22839.201,E2 -22839.201} C_VEL
LIN {X 0,Y 174.358,Z 679.318,A -85,B 0,C 180,E1 -22843.611,E2 -22843.611} C_VEL
LIN {X 0,Y 171.666,Z 676.711,A -85,B 0,C 180,E1 -22848.188,E2 -22848.188} C_VEL
LIN {X 0,Y 170.03,Z 672.915,A -85,B 0,C 180,E1 -22852.877,E2 -22852.877} C_VEL
LIN {X 0,Y 169.537,Z 667.829,A -85,B 0,C 180,E1 -22857.624,E2 -22857.624} C_VEL
LIN {X 0,Y 169.443,Z 662.979,A -85,B 0,C 180,E1 -22861.189,E2 -22861.189} C_VEL
LIN {X 0,Y 169.605,Z 655.755,A -85,B 0,C 180,E1 -22865.53,E2 -22865.53} C_VEL
LIN {X 0,Y 170.166,Z 647.622,A -85,B 0,C 180,E1 -22869.509,E2 -22869.509} C_VEL
LIN {X 0,Y 171.132,Z 637.27,A -85,B 0,C 180,E1 -22873.659,E2 -22873.659} C_VEL
LIN {X 0,Y 172.509,Z 626.59,A -85,B 0,C 180,E1 -22877.18,E2 -22877.18} C_VEL
LIN {X 0,Y 174.278,Z 613.685,A -85,B 0,C 180,E1 -22880.662,E2 -22880.662} C_VEL
LIN {X 0,Y 176.049,Z 601.557,A -85,B 0,C 180,E1 -22883.529,E2 -22883.529} C_VEL
LIN {X 0,Y 176.469,Z 600.48,A -85,B 0,C 180,E1 -22884.171,E2 -22884.171} C_VEL
LIN {X 0,Y 177.019,Z 600.419,A -85,B 0,C 180,E1 -22884.637,E2 -22884.637} C_VEL
LIN {X 0,Y 178.877,Z 599.332,A -85,B 0,C 180,E1 -22885.607,E2 -22885.607} C_VEL
LIN {X 0,Y 181.001,Z 597.239,A -85,B 0,C 180,E1 -22886.397,E2 -22886.397} C_VEL
LIN {X 0,Y 185.209,Z 592.061,A -85,B 0,C 180,E1 -22887.7,E2 -22887.7} C_VEL
LIN {X 0,Y 188.967,Z 589.409,A -85,B 0,C 180,E1 -22889.256,E2 -22889.256} C_VEL
LIN {X 0,Y 192.439,Z 585.145,A -85,B 0,C 180,E1 -22890.282,E2 -22890.282} C_VEL
LIN {X 0,Y 196.686,Z 578.122,A -85,B 0,C 180,E1 -22891.285,E2 -22891.285} C_VEL
LIN {X 0,Y 198.044,Z 575.934,A -85,B 0,C 180,E1 -22891.623,E2 -22891.623} C_VEL
LIN {X 0,Y 201.245,Z 572.404,A -85,B 0,C 180,E1 -22892.663,E2 -22892.663} C_VEL
LIN {X 0,Y 204.603,Z 567.14,A -85,B 0,C 180,E1 -22893.56,E2 -22893.56} C_VEL
LIN {X 0,Y 208.273,Z 558.746,A -85,B 0,C 180,E1 -22894.417,E2 -22894.417} C_VEL
LIN {X 0,Y 212.376,Z 545.966,A -85,B 0,C 180,E1 -22895.263,E2 -22895.263} C_VEL
LIN {X 0,Y 213.598,Z 541.94,A -85,B 0,C 180,E1 -22895.495,E2 -22895.495} C_VEL
LIN {X 0,Y 216.695,Z 536.811,A -85,B 0,C 180,E1 -22896.344,E2 -22896.344} C_VEL
LIN {X 0,Y 219.945,Z 529.288,A -85,B 0,C 180,E1 -22897.078,E2 -22897.078} C_VEL
LIN {X 0,Y 223.705,Z 518.501,A -85,B 0,C 180,E1 -22897.779,E2 -22897.779} C_VEL
LIN {X 0,Y 227.818,Z 504.982,A -85,B 0,C 180,E1 -22898.424,E2 -22898.424} C_VEL
LIN {X 0,Y 228.106,Z 504.544,A -85,B 0,C 180,E1 -22898.493,E2 -22898.493} C_VEL
LIN {X 0,Y 223.633,Z 565.169,A -85,B 0,C 180,E1 -22900.176,E2 -22900.176} C_VEL
LIN {X 0,Y 221.542,Z 580.421,A -85,B 0,C 180,E1 -22900.852,E2 -22900.852} C_VEL
LIN {X 0,Y 218.545,Z 595.214,A -85,B 0,C 180,E1 -22901.783,E2 -22901.783} C_VEL
LIN {X 0,Y 214.987,Z 609.098,A -85,B 0,C 180,E1 -22902.992,E2 -22902.992} C_VEL
LIN {X 0,Y 211.243,Z 621.324,A -85,B 0,C 180,E1 -22904.374,E2 -22904.374} C_VEL
LIN {X 0,Y 206.255,Z 635.166,A -85,B 0,C 180,E1 -22906.369,E2 -22906.369} C_VEL
LIN {X 0,Y 200.879,Z 647.814,A -85,B 0,C 180,E1 -22908.672,E2 -22908.672} C_VEL
LIN {X 0,Y 195.904,Z 658.41,A -85,B 0,C 180,E1 -22911.111,E2 -22911.111} C_VEL
LIN {X 0,Y 190.876,Z 668.212,A -85,B 0,C 180,E1 -22913.905,E2 -22913.905} C_VEL
LIN {X 0,Y 185.8,Z 677.795,A -85,B 0,C 180,E1 -22917.383,E2 -22917.383} C_VEL
LIN {X 0,Y 181.131,Z 685.777,A -85,B 0,C 180,E1 -22920.987,E2 -22920.987} C_VEL
LIN {X 0,Y 176.766,Z 693.208,A -85,B 0,C 180,E1 -22925.325,E2 -22925.325} C_VEL
LIN {X 0,Y 173.453,Z 699.104,A -85,B 0,C 180,E1 -22929.854,E2 -22929.854} C_VEL
LIN {X 0,Y 171.586,Z 702.589,A -85,B 0,C 180,E1 -22933.338,E2 -22933.338} C_VEL
LIN {X 0,Y 169.869,Z 706.14,A -85,B 0,C 180,E1 -22938.061,E2 -22938.061} C_VEL
LIN {X 0,Y 168.993,Z 708.482,A -85,B 0,C 180,E1 -22942.833,E2 -22942.833} C_VEL
LIN {X 0,Y 168.789,Z 709.669,A -85,B 0,C 180,E1 -22947.613,E2 -22947.613} C_VEL
LIN {X 0,Y 168.85,Z 709.825,A -85,B 0,C 180,E1 -22950,E2 -22950} C_VEL
LIN {X 0,Y 168.853,Z 709.247,A -85,B 0,C 180,E1 -22954.775,E2 -22954.775} C_VEL
LIN {X 0,Y 169.323,Z 707.527,A -85,B 0,C 180,E1 -22959.557,E2 -22959.557} C_VEL
LIN {X 0,Y 170.546,Z 704.635,A -85,B 0,C 180,E1 -22964.315,E2 -22964.315} C_VEL
LIN {X 0,Y 172.731,Z 700.502,A -85,B 0,C 180,E1 -22968.996,E2 -22968.996} C_VEL
LIN {X 0,Y 175.766,Z 695.015,A -85,B 0,C 180,E1 -22973.568,E2 -22973.568} C_VEL
LIN {X 0,Y 179.867,Z 688.027,A -85,B 0,C 180,E1 -22977.961,E2 -22977.961} C_VEL
LIN {X 0,Y 184.29,Z 680.546,A -85,B 0,C 180,E1 -22981.625,E2 -22981.625} C_VEL
LIN {X 0,Y 188.701,Z 672.453,A -85,B 0,C 180,E1 -22984.826,E2 -22984.826} C_VEL
LIN {X 0,Y 194.046,Z 662.32,A -85,B 0,C 180,E1 -22988.003,E2 -22988.003} C_VEL
LIN {X 0,Y 199.816,Z 650.456,A -85,B 0,C 180,E1 -22990.926,E2 -22990.926} C_VEL
LIN {X 0,Y 205.128,Z 638.347,A -85,B 0,C 180,E1 -22993.254,E2 -22993.254} C_VEL
LIN {X 0,Y 210.271,Z 624.726,A -85,B 0,C 180,E1 -22995.32,E2 -22995.32} C_VEL
LIN {X 0,Y 214.33,Z 611.959,A -85,B 0,C 180,E1 -22996.852,E2 -22996.852} C_VEL
LIN {X 0,Y 217.852,Z 598.782,A -85,B 0,C 180,E1 -22998.074,E2 -22998.074} C_VEL
LIN {X 0,Y 221.144,Z 583.701,A -85,B 0,C 180,E1 -22999.093,E2 -22999.093} C_VEL
LIN {X 0,Y 223.403,Z 568.883,A -85,B 0,C 180,E1 -22999.805,E2 -22999.805} C_VEL
LIN {X 0,Y 224.985,Z 550.888,A -85,B 0,C 180,E1 -23000.372,E2 -23000.372} C_VEL
LIN {X 0,Y 230.446,Z 474.959,A -85,B 0,C 180,E1 -23002.414,E2 -23002.414} C_VEL
LIN {X 0,Y 225.065,Z 462.258,A -85,B 0,C 180,E1 -23004.904,E2 -23004.904} C_VEL
LIN {X 0,Y 218.947,Z 449.932,A -85,B 0,C 180,E1 -23007.975,E2 -23007.975} C_VEL
LIN {X 0,Y 213.625,Z 440.503,A -85,B 0,C 180,E1 -23010.952,E2 -23010.952} C_VEL
LIN {X 0,Y 209.983,Z 434.743,A -85,B 0,C 180,E1 -23013.205,E2 -23013.205} C_VEL
LIN {X 0,Y 207.046,Z 430.109,A -85,B 0,C 180,E1 -23015.222,E2 -23015.222} C_VEL
LIN {X 0,Y 203.646,Z 425.033,A -85,B 0,C 180,E1 -23017.823,E2 -23017.823} C_VEL
LIN {X 0,Y 199.915,Z 419.725,A -85,B 0,C 180,E1 -23021.156,E2 -23021.156} C_VEL
LIN {X 0,Y 196.257,Z 414.825,A -85,B 0,C 180,E1 -23025.22,E2 -23025.22} C_VEL
LIN {X 0,Y 193.301,Z 410.922,A -85,B 0,C 180,E1 -23029.724,E2 -23029.724} C_VEL
LIN {X 0,Y 191.085,Z 408.037,A -85,B 0,C 180,E1 -23035.517,E2 -23035.517} C_VEL
LIN {X 0,Y 190.644,Z 406.533,A -85,B 0,C 180,E1 -23040,E2 -23040} C_VEL
LIN {X 0,Y 191.007,Z 407.476,A -85,B 0,C 180,E1 -23044.22,E2 -23044.22} C_VEL
LIN {X 0,Y 192.756,Z 409.898,A -85,B 0,C 180,E1 -23049.443,E2 -23049.443} C_VEL
LIN {X 0,Y 195.39,Z 412.736,A -85,B 0,C 180,E1 -23053.793,E2 -23053.793} C_VEL
LIN {X 0,Y 199.515,Z 417.886,A -85,B 0,C 180,E1 -23058.616,E2 -23058.616} C_VEL
LIN {X 0,Y 203.121,Z 422.637,A -85,B 0,C 180,E1 -23061.902,E2 -23061.902} C_VEL
LIN {X 0,Y 206.086,Z 426.681,A -85,B 0,C 180,E1 -23064.223,E2 -23064.223} C_VEL
LIN {X 0,Y 209.376,Z 431.392,A -85,B 0,C 180,E1 -23066.523,E2 -23066.523} C_VEL
LIN {X 0,Y 213.088,Z 436.728,A -85,B 0,C 180,E1 -23068.839,E2 -23068.839} C_VEL
LIN {X 0,Y 218.237,Z 444.744,A -85,B 0,C 180,E1 -23071.717,E2 -23071.717} C_VEL
LIN {X 0,Y 223.361,Z 453.565,A -85,B 0,C 180,E1 -23074.294,E2 -23074.294} C_VEL
LIN {X 0,Y 224.505,Z 456.524,A -85,B 0,C 180,E1 -23074.884,E2 -23074.884} C_VEL
LIN {X 0,Y 225.536,Z 461.744,A -85,B 0,C 180,E1 -23075.542,E2 -23075.542} C_VEL
LIN {X 0,Y 225.901,Z 467.447,A -85,B 0,C 180,E1 -23075.976,E2 -23075.976} C_VEL
LIN {X 0,Y 225.674,Z 475.601,A -85,B 0,C 180,E1 -23076.328,E2 -23076.328} C_VEL
LIN {X 0,Y 225.062,Z 483.827,A -85,B 0,C 180,E1 -23076.549,E2 -23076.549} C_VEL
LIN {X 0,Y 218.906,Z 564.969,A -85,B 0,C 180,E1 -23078.781,E2 -23078.781} C_VEL
LIN {X 0,Y 216.741,Z 580.282,A -85,B 0,C 180,E1 -23079.454,E2 -23079.454} C_VEL
LIN {X 0,Y 213.495,Z 595.712,A -85,B 0,C 180,E1 -23080.426,E2 -23080.426} C_VEL
LIN {X 0,Y 209.541,Z 610.391,A -85,B 0,C 180,E1 -23081.733,E2 -23081.733} C_VEL
LIN {X 0,Y 204.974,Z 624.491,A -85,B 0,C 180,E1 -23083.424,E2 -23083.424} C_VEL
LIN {X 0,Y 200.023,Z 637.196,A -85,B 0,C 180,E1 -23085.355,E2 -23085.355} C_VEL
LIN {X 0,Y 194.51,Z 649.434,A -85,B 0,C 180,E1 -23087.705,E2 -23087.705} C_VEL
LIN {X 0,Y 188.496,Z 661.41,A -85,B 0,C 180,E1 -23090.667,E2 -23090.667} C_VEL
LIN {X 0,Y 182.994,Z 671.283,A -85,B 0,C 180,E1 -23093.757,E2 -23093.757} C_VEL
LIN {X 0,Y 178.243,Z 679.743,A -85,B 0,C 180,E1 -23097.17,E2 -23097.17} C_VEL
LIN {X 0,Y 173.562,Z 687.269,A -85,B 0,C 180,E1 -23100.928,E2 -23100.928} C_VEL
LIN {X 0,Y 169.232,Z 694.292,A -85,B 0,C 180,E1 -23105.463,E2 -23105.463} C_VEL
LIN {X 0,Y 165.943,Z 699.806,A -85,B 0,C 180,E1 -23110.196,E2 -23110.196} C_VEL
LIN {X 0,Y 163.619,Z 703.96,A -85,B 0,C 180,E1 -23115.065,E2 -23115.065} C_VEL
LIN {X 0,Y 162.308,Z 706.868,A -85,B 0,C 180,E1 -23120.026,E2 -23120.026} C_VEL
LIN {X 0,Y 161.791,Z 708.6,A -85,B 0,C 180,E1 -23125.016,E2 -23125.016} C_VEL
LIN {X 0,Y 161.772,Z 709.188,A -85,B 0,C 180,E1 -23130,E2 -23130} C_VEL
LIN {X 0,Y 161.792,Z 708.588,A -85,B 0,C 180,E1 -23134.984,E2 -23134.984} C_VEL
LIN {X 0,Y 162.308,Z 706.839,A -85,B 0,C 180,E1 -23139.974,E2 -23139.974} C_VEL
LIN {X 0,Y 163.621,Z 703.908,A -85,B 0,C 180,E1 -23144.935,E2 -23144.935} C_VEL
LIN {X 0,Y 165.942,Z 699.727,A -85,B 0,C 180,E1 -23149.805,E2 -23149.805} C_VEL
LIN {X 0,Y 169.232,Z 694.194,A -85,B 0,C 180,E1 -23154.538,E2 -23154.538} C_VEL
LIN {X 0,Y 172.538,Z 689.275,A -85,B 0,C 180,E1 -23157.933,E2 -23157.933} C_VEL
LIN {X 0,Y 179.758,Z 687.485,A -85,B 0,C 180,E1 -23163.186,E2 -23163.186} C_VEL
LIN {X 0,Y 186.874,Z 685.177,A -85,B 0,C 180,E1 -23166.994,E2 -23166.994} C_VEL
LIN {X 0,Y 194.99,Z 682,A -85,B 0,C 180,E1 -23170.449,E2 -23170.449} C_VEL
LIN {X 0,Y 206.569,Z 676.841,A -85,B 0,C 180,E1 -23174.224,E2 -23174.224} C_VEL
LIN {X 0,Y 216.337,Z 671.94,A -85,B 0,C 180,E1 -23176.781,E2 -23176.781} C_VEL
LIN {X 0,Y 218.183,Z 670.889,A -85,B 0,C 180,E1 -23177.434,E2 -23177.434} C_VEL
LIN {X 0,Y 208.192,Z 675.042,A -85,B 0,C 180,E1 -23180.105,E2 -23180.105} C_VEL
LIN {X 0,Y 198.942,Z 678.232,A -85,B 0,C 180,E1 -23183.09,E2 -23183.09} C_VEL
LIN {X 0,Y 190.424,Z 680.462,A -85,B 0,C 180,E1 -23186.386,E2 -23186.386} C_VEL
LIN {X 0,Y 183.045,Z 681.626,A -85,B 0,C 180,E1 -23190.058,E2 -23190.058} C_VEL
LIN {X 0,Y 176.653,Z 681.83,A -85,B 0,C 180,E1 -23194.048,E2 -23194.048} C_VEL
LIN {X 0,Y 171.51,Z 681.038,A -85,B 0,C 180,E1 -23198.359,E2 -23198.359} C_VEL
LIN {X 0,Y 167.558,Z 679.196,A -85,B 0,C 180,E1 -23202.926,E2 -23202.926} C_VEL
LIN {X 0,Y 164.749,Z 676.239,A -85,B 0,C 180,E1 -23207.685,E2 -23207.685} C_VEL
LIN {X 0,Y 163.054,Z 672.113,A -85,B 0,C 180,E1 -23212.571,E2 -23212.571} C_VEL
LIN {X 0,Y 162.545,Z 666.712,A -85,B 0,C 180,E1 -23217.522,E2 -23217.522} C_VEL
LIN {X 0,Y 162.432,Z 661.647,A -85,B 0,C 180,E1 -23221.24,E2 -23221.24} C_VEL
LIN {X 0,Y 162.613,Z 654.419,A -85,B 0,C 180,E1 -23225.581,E2 -23225.581} C_VEL
LIN {X 0,Y 163.13,Z 646.957,A -85,B 0,C 180,E1 -23229.298,E2 -23229.298} C_VEL
LIN {X 0,Y 164.113,Z 636.398,A -85,B 0,C 180,E1 -23233.623,E2 -23233.623} C_VEL
LIN {X 0,Y 165.49,Z 625.525,A -85,B 0,C 180,E1 -23237.294,E2 -23237.294} C_VEL
LIN {X 0,Y 167.109,Z 613.882,A -85,B 0,C 180,E1 -23240.624,E2 -23240.624} C_VEL
LIN {X 0,Y 167.571,Z 612.185,A -85,B 0,C 180,E1 -23241.53,E2 -23241.53} C_VEL
LIN {X 0,Y 168.073,Z 612.091,A -85,B 0,C 180,E1 -23242.107,E2 -23242.107} C_VEL
LIN {X 0,Y 169.876,Z 611.263,A -85,B 0,C 180,E1 -23243.226,E2 -23243.226} C_VEL
LIN {X 0,Y 173.172,Z 608.336,A -85,B 0,C 180,E1 -23244.582,E2 -23244.582} C_VEL
LIN {X 0,Y 174.488,Z 606.94,A -85,B 0,C 180,E1 -23245.019,E2 -23245.019} C_VEL
LIN {X 0,Y 176.29,Z 606.23,A -85,B 0,C 180,E1 -23246.01,E2 -23246.01} C_VEL
LIN {X 0,Y 178.358,Z 605.005,A -85,B 0,C 180,E1 -23246.952,E2 -23246.952} C_VEL
LIN {X 0,Y 180.796,Z 602.788,A -85,B 0,C 180,E1 -23247.806,E2 -23247.806} C_VEL
LIN {X 0,Y 184.561,Z 598.49,A -85,B 0,C 180,E1 -23248.856,E2 -23248.856} C_VEL
LIN {X 0,Y 189.525,Z 594.755,A -85,B 0,C 180,E1 -23250.656,E2 -23250.656} C_VEL
LIN {X 0,Y 193.647,Z 590.124,A -85,B 0,C 180,E1 -23251.752,E2 -23251.752} C_VEL
LIN {X 0,Y 198.174,Z 583.387,A -85,B 0,C 180,E1 -23252.73,E2 -23252.73} C_VEL
LIN {X 0,Y 199.708,Z 580.945,A -85,B 0,C 180,E1 -23253.057,E2 -23253.057} C_VEL
LIN {X 0,Y 203.581,Z 576.641,A -85,B 0,C 180,E1 -23254.153,E2 -23254.153} C_VEL
LIN {X 0,Y 207.333,Z 570.93,A -85,B 0,C 180,E1 -23255.048,E2 -23255.048} C_VEL
LIN {X 0,Y 211.193,Z 562.774,A -85,B 0,C 180,E1 -23255.837,E2 -23255.837} C_VEL
LIN {X 0,Y 215.466,Z 550.407,A -85,B 0,C 180,E1 -23256.649,E2 -23256.649} C_VEL
LIN {X 0,Y 216.902,Z 545.729,A -85,B 0,C 180,E1 -23256.902,E2 -23256.902} C_VEL
LIN {X 0,Y 220.475,Z 539.544,A -85,B 0,C 180,E1 -23257.796,E2 -23257.796} C_VEL
LIN {X 0,Y 221.28,Z 537.807,A -85,B 0,C 180,E1 -23257.973,E2 -23257.973} C_VEL
LIN {X 0,Y 219.022,Z 566.093,A -85,B 0,C 180,E1 -23258.792,E2 -23258.792} C_VEL
LIN {X 0,Y 216.665,Z 582.108,A -85,B 0,C 180,E1 -23259.52,E2 -23259.52} C_VEL
LIN {X 0,Y 213.299,Z 597.619,A -85,B 0,C 180,E1 -23260.545,E2 -23260.545} C_VEL
LIN {X 0,Y 209.64,Z 611.009,A -85,B 0,C 180,E1 -23261.762,E2 -23261.762} C_VEL
LIN {X 0,Y 205.409,Z 624.03,A -85,B 0,C 180,E1 -23263.319,E2 -23263.319} C_VEL
LIN {X 0,Y 200.621,Z 636.415,A -85,B 0,C 180,E1 -23265.17,E2 -23265.17} C_VEL
LIN {X 0,Y 195.101,Z 648.85,A -85,B 0,C 180,E1 -23267.513,E2 -23267.513} C_VEL
LIN {X 0,Y 189.487,Z 660.153,A -85,B 0,C 180,E1 -23270.223,E2 -23270.223} C_VEL
LIN {X 0,Y 184.411,Z 669.516,A -85,B 0,C 180,E1 -23273.044,E2 -23273.044} C_VEL
LIN {X 0,Y 179.073,Z 678.998,A -85,B 0,C 180,E1 -23276.67,E2 -23276.67} C_VEL
LIN {X 0,Y 174.897,Z 685.762,A -85,B 0,C 180,E1 -23279.848,E2 -23279.848} C_VEL
LIN {X 0,Y 170.293,Z 693.194,A -85,B 0,C 180,E1 -23284.32,E2 -23284.32} C_VEL
LIN {X 0,Y 166.755,Z 699.091,A -85,B 0,C 180,E1 -23289.008,E2 -23289.008} C_VEL
LIN {X 0,Y 164.766,Z 702.575,A -85,B 0,C 180,E1 -23292.627,E2 -23292.627} C_VEL
LIN {X 0,Y 162.872,Z 706.127,A -85,B 0,C 180,E1 -23297.54,E2 -23297.54} C_VEL
LIN {X 0,Y 161.931,Z 708.468,A -85,B 0,C 180,E1 -23302.518,E2 -23302.518} C_VEL
LIN {X 0,Y 161.713,Z 709.655,A -85,B 0,C 180,E1 -23307.509,E2 -23307.509} C_VEL
LIN {X 0,Y 161.773,Z 709.811,A -85,B 0,C 180,E1 -23310,E2 -23310} C_VEL
LIN {X 0,Y 161.755,Z 709.233,A -85,B 0,C 180,E1 -23314.985,E2 -23314.985} C_VEL
LIN {X 0,Y 162.31,Z 707.513,A -85,B 0,C 180,E1 -23319.974,E2 -23319.974} C_VEL
LIN {X 0,Y 163.625,Z 704.62,A -85,B 0,C 180,E1 -23324.934,E2 -23324.934} C_VEL
LIN {X 0,Y 165.965,Z 700.486,A -85,B 0,C 180,E1 -23329.802,E2 -23329.802} C_VEL
LIN {X 0,Y 169.236,Z 694.998,A -85,B 0,C 180,E1 -23334.537,E2 -23334.537} C_VEL
LIN {X 0,Y 173.57,Z 688.01,A -85,B 0,C 180,E1 -23339.07,E2 -23339.07} C_VEL
LIN {X 0,Y 178.25,Z 680.527,A -85,B 0,C 180,E1 -23342.829,E2 -23342.829} C_VEL
LIN {X 0,Y 183.191,Z 671.849,A -85,B 0,C 180,E1 -23346.326,E2 -23346.326} C_VEL
LIN {X 0,Y 188.48,Z 662.299,A -85,B 0,C 180,E1 -23349.338,E2 -23349.338} C_VEL
LIN {X 0,Y 194.486,Z 650.432,A -85,B 0,C 180,E1 -23352.302,E2 -23352.302} C_VEL
LIN {X 0,Y 200.011,Z 638.319,A -85,B 0,C 180,E1 -23354.649,E2 -23354.649} C_VEL
LIN {X 0,Y 205.053,Z 625.437,A -85,B 0,C 180,E1 -23356.635,E2 -23356.635} C_VEL
LIN {X 0,Y 209.539,Z 611.92,A -85,B 0,C 180,E1 -23358.268,E2 -23358.268} C_VEL
LIN {X 0,Y 213.18,Z 598.735,A -85,B 0,C 180,E1 -23359.491,E2 -23359.491} C_VEL
LIN {X 0,Y 216.418,Z 584.372,A -85,B 0,C 180,E1 -23360.467,E2 -23360.467} C_VEL
LIN {X 0,Y 218.747,Z 569.87,A -85,B 0,C 180,E1 -23361.179,E2 -23361.179} C_VEL
LIN {X 0,Y 220.4,Z 552.528,A -85,B 0,C 180,E1 -23361.742,E2 -23361.742} C_VEL
LIN {X 0,Y 225.964,Z 477.469,A -85,B 0,C 180,E1 -23363.776,E2 -23363.776} C_VEL
LIN {X 0,Y 220.859,Z 465.421,A -85,B 0,C 180,E1 -23366.297,E2 -23366.297} C_VEL
LIN {X 0,Y 215.472,Z 454.398,A -85,B 0,C 180,E1 -23369.19,E2 -23369.19} C_VEL
LIN {X 0,Y 210.458,Z 445.231,A -85,B 0,C 180,E1 -23372.194,E2 -23372.194} C_VEL
LIN {X 0,Y 205.28,Z 436.8,A -85,B 0,C 180,E1 -23375.743,E2 -23375.743} C_VEL
LIN {X 0,Y 201.631,Z 431.196,A -85,B 0,C 180,E1 -23378.666,E2 -23378.666} C_VEL
LIN {X 0,Y 198.185,Z 426.156,A -85,B 0,C 180,E1 -23381.923,E2 -23381.923} C_VEL
LIN {X 0,Y 195.005,Z 421.63,A -85,B 0,C 180,E1 -23385.654,E2 -23385.654} C_VEL
LIN {X 0,Y 192.229,Z 417.845,A -85,B 0,C 180,E1 -23390.065,E2 -23390.065} C_VEL
LIN {X 0,Y 190.062,Z 414.795,A -85,B 0,C 180,E1 -23396.29,E2 -23396.29} C_VEL
LIN {X 0,Y 189.779,Z 413.574,A -85,B 0,C 180,E1 -23400,E2 -23400} C_VEL
LIN {X 0,Y 190.141,Z 414.55,A -85,B 0,C 180,E1 -23404.239,E2 -23404.239} C_VEL
LIN {X 0,Y 191.893,Z 417.025,A -85,B 0,C 180,E1 -23409.486,E2 -23409.486} C_VEL
LIN {X 0,Y 194.217,Z 419.647,A -85,B 0,C 180,E1 -23413.423,E2 -23413.423} C_VEL
LIN {X 0,Y 197.852,Z 424.347,A -85,B 0,C 180,E1 -23417.884,E2 -23417.884} C_VEL
LIN {X 0,Y 201.375,Z 429.151,A -85,B 0,C 180,E1 -23421.262,E2 -23421.262} C_VEL
LIN {X 0,Y 204.207,Z 433.181,A -85,B 0,C 180,E1 -23423.583,E2 -23423.583} C_VEL
LIN {X 0,Y 207.107,Z 437.4,A -85,B 0,C 180,E1 -23425.704,E2 -23425.704} C_VEL
LIN {X 0,Y 210.758,Z 442.886,A -85,B 0,C 180,E1 -23428.1,E2 -23428.1} C_VEL
LIN {X 0,Y 214.682,Z 449.154,A -85,B 0,C 180,E1 -23430.424,E2 -23430.424} C_VEL
LIN {X 0,Y 219.947,Z 458.344,A -85,B 0,C 180,E1 -23433.24,E2 -23433.24} C_VEL
LIN {X 0,Y 223.586,Z 465.424,A -85,B 0,C 180,E1 -23435.035,E2 -23435.035} C_VEL
LIN {X 0,Y 225.878,Z 472.576,A -85,B 0,C 180,E1 -23436.24,E2 -23436.24} C_VEL
LIN {X 0,Y 225.062,Z 483.827,A -85,B 0,C 180,E1 -23436.549,E2 -23436.549} C_VEL
LIN {X 0,Y 224.21,Z 489.678,A -85,B 0,C 180,E1 -23436.563,E2 -23436.563} C_VEL
LIN {X 0,Y 219.389,Z 508.74,A -85,B 0,C 180,E1 -23435.879,E2 -23435.879} C_VEL
LIN {X 0,Y 218.559,Z 514.589,A -85,B 0,C 180,E1 -23435.898,E2 -23435.898} C_VEL
LIN {X 0,Y 214.547,Z 565.084,A -85,B 0,C 180,E1 -23437.308,E2 -23437.308} C_VEL
LIN {X 0,Y 212.308,Z 580.354,A -85,B 0,C 180,E1 -23437.977,E2 -23437.977} C_VEL
LIN {X 0,Y 208.975,Z 595.764,A -85,B 0,C 180,E1 -23438.949,E2 -23438.949} C_VEL
LIN {X 0,Y 204.882,Z 610.431,A -85,B 0,C 180,E1 -23440.25,E2 -23440.25} C_VEL
LIN {X 0,Y 200.136,Z 624.524,A -85,B 0,C 180,E1 -23441.94,E2 -23441.94} C_VEL
LIN {X 0,Y 195.029,Z 637.224,A -85,B 0,C 180,E1 -23443.887,E2 -23443.887} C_VEL
LIN {X 0,Y 189.304,Z 649.459,A -85,B 0,C 180,E1 -23446.254,E2 -23446.254} C_VEL
LIN {X 0,Y 183.031,Z 661.431,A -85,B 0,C 180,E1 -23449.25,E2 -23449.25} C_VEL
LIN {X 0,Y 176.965,Z 671.823,A -85,B 0,C 180,E1 -23452.587,E2 -23452.587} C_VEL
LIN {X 0,Y 172.288,Z 679.762,A -85,B 0,C 180,E1 -23455.883,E2 -23455.883} C_VEL
LIN {X 0,Y 167.356,Z 687.287,A -85,B 0,C 180,E1 -23459.74,E2 -23459.74} C_VEL
LIN {X 0,Y 162.759,Z 694.309,A -85,B 0,C 180,E1 -23464.418,E2 -23464.418} C_VEL
LIN {X 0,Y 159.22,Z 699.821,A -85,B 0,C 180,E1 -23469.322,E2 -23469.322} C_VEL
LIN {X 0,Y 156.717,Z 703.975,A -85,B 0,C 180,E1 -23474.391,E2 -23474.391} C_VEL
LIN {X 0,Y 155.278,Z 706.882,A -85,B 0,C 180,E1 -23479.57,E2 -23479.57} C_VEL
LIN {X 0,Y 154.707,Z 708.614,A -85,B 0,C 180,E1 -23484.788,E2 -23484.788} C_VEL
LIN {X 0,Y 154.684,Z 709.201,A -85,B 0,C 180,E1 -23490,E2 -23490} C_VEL
LIN {X 0,Y 154.707,Z 708.602,A -85,B 0,C 180,E1 -23495.213,E2 -23495.213} C_VEL
LIN {X 0,Y 155.279,Z 706.853,A -85,B 0,C 180,E1 -23500.431,E2 -23500.431} C_VEL
LIN {X 0,Y 156.721,Z 703.922,A -85,B 0,C 180,E1 -23505.609,E2 -23505.609} C_VEL
LIN {X 0,Y 159.22,Z 699.741,A -85,B 0,C 180,E1 -23510.679,E2 -23510.679} C_VEL
LIN {X 0,Y 162.761,Z 694.208,A -85,B 0,C 180,E1 -23515.582,E2 -23515.582} C_VEL
LIN {X 0,Y 166.592,Z 688.882,A -85,B 0,C 180,E1 -23519.369,E2 -23519.369} C_VEL
LIN {X 0,Y 173.859,Z 687.56,A -85,B 0,C 180,E1 -23524.467,E2 -23524.467} C_VEL
LIN {X 0,Y 185.32,Z 684.351,A -85,B 0,C 180,E1 -23530.144,E2 -23530.144} C_VEL
LIN {X 0,Y 194.33,Z 681.148,A -85,B 0,C 180,E1 -23533.405,E2 -23533.405} C_VEL
LIN {X 0,Y 204.175,Z 677.198,A -85,B 0,C 180,E1 -23536.291,E2 -23536.291} C_VEL
LIN {X 0,Y 208.053,Z 675.42,A -85,B 0,C 180,E1 -23537.5,E2 -23537.5} C_VEL
LIN {X 0,Y 198.16,Z 678.623,A -85,B 0,C 180,E1 -23540.328,E2 -23540.328} C_VEL
LIN {X 0,Y 188.951,Z 680.864,A -85,B 0,C 180,E1 -23543.479,E2 -23543.479} C_VEL
LIN {X 0,Y 180.683,Z 682.136,A -85,B 0,C 180,E1 -23547.006,E2 -23547.006} C_VEL
LIN {X 0,Y 173.531,Z 682.47,A -85,B 0,C 180,E1 -23550.922,E2 -23550.922} C_VEL
LIN {X 0,Y 167.442,Z 681.81,A -85,B 0,C 180,E1 -23555.183,E2 -23555.183} C_VEL
LIN {X 0,Y 162.726,Z 680.119,A -85,B 0,C 180,E1 -23559.787,E2 -23559.787} C_VEL
LIN {X 0,Y 159.146,Z 677.406,A -85,B 0,C 180,E1 -23564.635,E2 -23564.635} C_VEL
LIN {X 0,Y 156.785,Z 673.577,A -85,B 0,C 180,E1 -23569.671,E2 -23569.671} C_VEL
LIN {X 0,Y 155.76,Z 668.543,A -85,B 0,C 180,E1 -23574.823,E2 -23574.823} C_VEL
LIN {X 0,Y 155.503,Z 663.803,A -85,B 0,C 180,E1 -23578.705,E2 -23578.705} C_VEL
LIN {X 0,Y 155.473,Z 657.064,A -85,B 0,C 180,E1 -23583.24,E2 -23583.24} C_VEL
LIN {X 0,Y 155.886,Z 648.807,A -85,B 0,C 180,E1 -23587.774,E2 -23587.774} C_VEL
LIN {X 0,Y 156.74,Z 638.709,A -85,B 0,C 180,E1 -23592.298,E2 -23592.298} C_VEL
LIN {X 0,Y 157.982,Z 628.299,A -85,B 0,C 180,E1 -23596.143,E2 -23596.143} C_VEL
LIN {X 0,Y 158.693,Z 622.828,A -85,B 0,C 180,E1 -23598.06,E2 -23598.06} C_VEL
LIN {X 0,Y 158.915,Z 622.143,A -85,B 0,C 180,E1 -23598.701,E2 -23598.701} C_VEL
LIN {X 0,Y 159.343,Z 622.141,A -85,B 0,C 180,E1 -23599.317,E2 -23599.317} C_VEL
LIN {X 0,Y 160.814,Z 621.606,A -85,B 0,C 180,E1 -23600.464,E2 -23600.464} C_VEL
LIN {X 0,Y 165.079,Z 618.41,A -85,B 0,C 180,E1 -23602.53,E2 -23602.53} C_VEL
LIN {X 0,Y 168.634,Z 616.869,A -85,B 0,C 180,E1 -23604.631,E2 -23604.631} C_VEL
LIN {X 0,Y 171.894,Z 614.286,A -85,B 0,C 180,E1 -23605.909,E2 -23605.909} C_VEL
LIN {X 0,Y 173.545,Z 612.797,A -85,B 0,C 180,E1 -23606.453,E2 -23606.453} C_VEL
LIN {X 0,Y 177.736,Z 610.618,A -85,B 0,C 180,E1 -23608.327,E2 -23608.327} C_VEL
LIN {X 0,Y 181.212,Z 607.635,A -85,B 0,C 180,E1 -23609.441,E2 -23609.441} C_VEL
LIN {X 0,Y 184.591,Z 604.165,A -85,B 0,C 180,E1 -23610.297,E2 -23610.297} C_VEL
LIN {X 0,Y 185.876,Z 603.043,A -85,B 0,C 180,E1 -23610.693,E2 -23610.693} C_VEL
LIN {X 0,Y 188.203,Z 601.564,A -85,B 0,C 180,E1 -23611.52,E2 -23611.52} C_VEL
LIN {X 0,Y 191.636,Z 598.554,A -85,B 0,C 180,E1 -23612.488,E2 -23612.488} C_VEL
LIN {X 0,Y 196.713,Z 592.639,A -85,B 0,C 180,E1 -23613.626,E2 -23613.626} C_VEL
LIN {X 0,Y 201.427,Z 585.787,A -85,B 0,C 180,E1 -23614.499,E2 -23614.499} C_VEL
LIN {X 0,Y 205.581,Z 581.346,A -85,B 0,C 180,E1 -23615.533,E2 -23615.533} C_VEL
LIN {X 0,Y 210.107,Z 574.857,A -85,B 0,C 180,E1 -23616.482,E2 -23616.482} C_VEL
LIN {X 0,Y 214.608,Z 565.864,A -85,B 0,C 180,E1 -23617.291,E2 -23617.291} C_VEL
LIN {X 0,Y 212.468,Z 580.763,A -85,B 0,C 180,E1 -23617.983,E2 -23617.983} C_VEL
LIN {X 0,Y 209.295,Z 595.425,A -85,B 0,C 180,E1 -23618.908,E2 -23618.908} C_VEL
LIN {X 0,Y 205.565,Z 609.042,A -85,B 0,C 180,E1 -23620.095,E2 -23620.095} C_VEL
LIN {X 0,Y 201.234,Z 622.066,A -85,B 0,C 180,E1 -23621.573,E2 -23621.573} C_VEL
LIN {X 0,Y 196.218,Z 635.125,A -85,B 0,C 180,E1 -23623.506,E2 -23623.506} C_VEL
LIN {X 0,Y 190.391,Z 647.777,A -85,B 0,C 180,E1 -23625.833,E2 -23625.833} C_VEL
LIN {X 0,Y 185.007,Z 658.376,A -85,B 0,C 180,E1 -23628.334,E2 -23628.334} C_VEL
LIN {X 0,Y 179.526,Z 668.18,A -85,B 0,C 180,E1 -23631.217,E2 -23631.217} C_VEL
LIN {X 0,Y 174.699,Z 676.535,A -85,B 0,C 180,E1 -23634.315,E2 -23634.315} C_VEL
LIN {X 0,Y 169.39,Z 684.702,A -85,B 0,C 180,E1 -23638.062,E2 -23638.062} C_VEL
LIN {X 0,Y 164.988,Z 691.461,A -85,B 0,C 180,E1 -23642.058,E2 -23642.058} C_VEL
LIN {X 0,Y 160.939,Z 697.719,A -85,B 0,C 180,E1 -23646.857,E2 -23646.857} C_VEL
LIN {X 0,Y 157.943,Z 702.562,A -85,B 0,C 180,E1 -23651.851,E2 -23651.851} C_VEL
LIN {X 0,Y 155.901,Z 706.113,A -85,B 0,C 180,E1 -23656.973,E2 -23656.973} C_VEL
LIN {X 0,Y 154.87,Z 708.455,A -85,B 0,C 180,E1 -23662.175,E2 -23662.175} C_VEL
LIN {X 0,Y 154.629,Z 709.641,A -85,B 0,C 180,E1 -23667.395,E2 -23667.395} C_VEL
LIN {X 0,Y 154.641,Z 709.749,A -85,B 0,C 180,E1 -23671.007,E2 -23671.007} C_VEL
LIN {X 0,Y 154.684,Z 709.219,A -85,B 0,C 180,E1 -23675.213,E2 -23675.213} C_VEL
LIN {X 0,Y 155.28,Z 707.498,A -85,B 0,C 180,E1 -23680.43,E2 -23680.43} C_VEL
LIN {X 0,Y 156.723,Z 704.605,A -85,B 0,C 180,E1 -23685.608,E2 -23685.608} C_VEL
LIN {X 0,Y 159.241,Z 700.47,A -85,B 0,C 180,E1 -23690.675,E2 -23690.675} C_VEL
LIN {X 0,Y 162.764,Z 694.982,A -85,B 0,C 180,E1 -23695.581,E2 -23695.581} C_VEL
LIN {X 0,Y 167.346,Z 687.992,A -85,B 0,C 180,E1 -23700.262,E2 -23700.262} C_VEL
LIN {X 0,Y 172.295,Z 680.508,A -85,B 0,C 180,E1 -23704.116,E2 -23704.116} C_VEL
LIN {X 0,Y 177.765,Z 671.393,A -85,B 0,C 180,E1 -23707.839,E2 -23707.839} C_VEL
LIN {X 0,Y 183.01,Z 662.277,A -85,B 0,C 180,E1 -23710.756,E2 -23710.756} C_VEL
LIN {X 0,Y 189.252,Z 650.407,A -85,B 0,C 180,E1 -23713.761,E2 -23713.761} C_VEL
LIN {X 0,Y 195.016,Z 638.291,A -85,B 0,C 180,E1 -23716.117,E2 -23716.117} C_VEL
LIN {X 0,Y 199.925,Z 626.17,A -85,B 0,C 180,E1 -23718.009,E2 -23718.009} C_VEL
LIN {X 0,Y 204.865,Z 611.882,A -85,B 0,C 180,E1 -23719.756,E2 -23719.756} C_VEL
LIN {X 0,Y 208.927,Z 597.591,A -85,B 0,C 180,E1 -23721.068,E2 -23721.068} C_VEL
LIN {X 0,Y 212.267,Z 582.842,A -85,B 0,C 180,E1 -23722.037,E2 -23722.037} C_VEL
LIN {X 0,Y 214.659,Z 567.625,A -85,B 0,C 180,E1 -23722.75,E2 -23722.75} C_VEL
LIN {X 0,Y 216.752,Z 543.442,A -85,B 0,C 180,E1 -23723.467,E2 -23723.467} C_VEL
LIN {X 0,Y 221.598,Z 480.131,A -85,B 0,C 180,E1 -23725.189,E2 -23725.189} C_VEL
LIN {X 0,Y 217.317,Z 469.813,A -85,B 0,C 180,E1 -23727.451,E2 -23727.451} C_VEL
LIN {X 0,Y 212.61,Z 459.848,A -85,B 0,C 180,E1 -23730.138,E2 -23730.138} C_VEL
LIN {X 0,Y 207.736,Z 450.693,A -85,B 0,C 180,E1 -23733.232,E2 -23733.232} C_VEL
LIN {X 0,Y 203.089,Z 442.789,A -85,B 0,C 180,E1 -23736.616,E2 -23736.616} C_VEL
LIN {X 0,Y 199.793,Z 437.552,A -85,B 0,C 180,E1 -23739.405,E2 -23739.405} C_VEL
LIN {X 0,Y 196.608,Z 432.711,A -85,B 0,C 180,E1 -23742.58,E2 -23742.58} C_VEL
LIN {X 0,Y 193.484,Z 428.106,A -85,B 0,C 180,E1 -23746.477,E2 -23746.477} C_VEL
LIN {X 0,Y 191.009,Z 424.54,A -85,B 0,C 180,E1 -23750.736,E2 -23750.736} C_VEL
LIN {X 0,Y 189.071,Z 421.578,A -85,B 0,C 180,E1 -23757.07,E2 -23757.07} C_VEL
LIN {X 0,Y 188.914,Z 420.622,A -85,B 0,C 180,E1 -23760,E2 -23760} C_VEL
LIN {X 0,Y 189.275,Z 421.626,A -85,B 0,C 180,E1 -23764.259,E2 -23764.259} C_VEL
LIN {X 0,Y 191.025,Z 424.2,A -85,B 0,C 180,E1 -23769.53,E2 -23769.53} C_VEL
LIN {X 0,Y 193.035,Z 426.515,A -85,B 0,C 180,E1 -23773.019,E2 -23773.019} C_VEL
LIN {X 0,Y 196.505,Z 431.206,A -85,B 0,C 180,E1 -23777.456,E2 -23777.456} C_VEL
LIN {X 0,Y 199.721,Z 435.758,A -85,B 0,C 180,E1 -23780.67,E2 -23780.67} C_VEL
LIN {X 0,Y 202.435,Z 439.775,A -85,B 0,C 180,E1 -23782.995,E2 -23782.995} C_VEL
LIN {X 0,Y 204.914,Z 443.494,A -85,B 0,C 180,E1 -23784.894,E2 -23784.894} C_VEL
LIN {X 0,Y 208.675,Z 449.346,A -85,B 0,C 180,E1 -23787.48,E2 -23787.48} C_VEL
LIN {X 0,Y 213.004,Z 456.579,A -85,B 0,C 180,E1 -23790.135,E2 -23790.135} C_VEL
LIN {X 0,Y 218.093,Z 465.986,A -85,B 0,C 180,E1 -23792.942,E2 -23792.942} C_VEL
LIN {X 0,Y 220.178,Z 470.369,A -85,B 0,C 180,E1 -23794.026,E2 -23794.026} C_VEL
LIN {X 0,Y 221.574,Z 474.93,A -85,B 0,C 180,E1 -23794.815,E2 -23794.815} C_VEL
LIN {X 0,Y 218.559,Z 514.589,A -85,B 0,C 180,E1 -23795.898,E2 -23795.898} C_VEL
LIN {X 0,Y 217.725,Z 520.44,A -85,B 0,C 180,E1 -23795.917,E2 -23795.917} C_VEL
LIN {X 0,Y 212.926,Z 539.508,A -85,B 0,C 180,E1 -23795.194,E2 -23795.194} C_VEL
LIN {X 0,Y 212.089,Z 545.36,A -85,B 0,C 180,E1 -23795.209,E2 -23795.209} C_VEL
LIN {X 0,Y 209.995,Z 567.667,A -85,B 0,C 180,E1 -23795.852,E2 -23795.852} C_VEL
LIN {X 0,Y 207.561,Z 582.841,A -85,B 0,C 180,E1 -23796.572,E2 -23796.572} C_VEL
LIN {X 0,Y 204.285,Z 596.999,A -85,B 0,C 180,E1 -23797.494,E2 -23797.494} C_VEL
LIN {X 0,Y 200.368,Z 610.471,A -85,B 0,C 180,E1 -23798.701,E2 -23798.701} C_VEL
LIN {X 0,Y 195.329,Z 624.895,A -85,B 0,C 180,E1 -23800.44,E2 -23800.44} C_VEL
LIN {X 0,Y 189.618,Z 638.438,A -85,B 0,C 180,E1 -23802.554,E2 -23802.554} C_VEL
LIN {X 0,Y 183.7,Z 650.472,A -85,B 0,C 180,E1 -23804.946,E2 -23804.946} C_VEL
LIN {X 0,Y 177.702,Z 661.453,A -85,B 0,C 180,E1 -23807.752,E2 -23807.752} C_VEL
LIN {X 0,Y 171.899,Z 671.005,A -85,B 0,C 180,E1 -23810.827,E2 -23810.827} C_VEL
LIN {X 0,Y 166.418,Z 679.78,A -85,B 0,C 180,E1 -23814.502,E2 -23814.502} C_VEL
LIN {X 0,Y 161.235,Z 687.304,A -85,B 0,C 180,E1 -23818.463,E2 -23818.463} C_VEL
LIN {X 0,Y 156.336,Z 694.325,A -85,B 0,C 180,E1 -23823.286,E2 -23823.286} C_VEL
LIN {X 0,Y 152.545,Z 699.837,A -85,B 0,C 180,E1 -23828.373,E2 -23828.373} C_VEL
LIN {X 0,Y 149.839,Z 703.99,A -85,B 0,C 180,E1 -23833.655,E2 -23833.655} C_VEL
LIN {X 0,Y 148.271,Z 706.896,A -85,B 0,C 180,E1 -23839.071,E2 -23839.071} C_VEL
LIN {X 0,Y 147.626,Z 708.628,A -85,B 0,C 180,E1 -23844.537,E2 -23844.537} C_VEL
LIN {X 0,Y 147.587,Z 709.215,A -85,B 0,C 180,E1 -23850,E2 -23850} C_VEL
LIN {X 0,Y 147.626,Z 708.615,A -85,B 0,C 180,E1 -23855.464,E2 -23855.464} C_VEL
LIN {X 0,Y 148.272,Z 706.866,A -85,B 0,C 180,E1 -23860.93,E2 -23860.93} C_VEL
LIN {X 0,Y 149.843,Z 703.935,A -85,B 0,C 180,E1 -23866.345,E2 -23866.345} C_VEL
LIN {X 0,Y 152.545,Z 699.754,A -85,B 0,C 180,E1 -23871.628,E2 -23871.628} C_VEL
LIN {X 0,Y 156.339,Z 694.222,A -85,B 0,C 180,E1 -23876.714,E2 -23876.714} C_VEL
LIN {X 0,Y 160.783,Z 688.403,A -85,B 0,C 180,E1 -23880.905,E2 -23880.905} C_VEL
LIN {X 0,Y 168.033,Z 687.516,A -85,B 0,C 180,E1 -23885.842,E2 -23885.842} C_VEL
LIN {X 0,Y 179.966,Z 684.822,A -85,B 0,C 180,E1 -23891.597,E2 -23891.597} C_VEL
LIN {X 0,Y 189.278,Z 682.076,A -85,B 0,C 180,E1 -23894.869,E2 -23894.869} C_VEL
LIN {X 0,Y 194.273,Z 680.394,A -85,B 0,C 180,E1 -23896.346,E2 -23896.346} C_VEL
LIN {X 0,Y 197.892,Z 679.09,A -85,B 0,C 180,E1 -23897.564,E2 -23897.564} C_VEL
LIN {X 0,Y 188.03,Z 681.323,A -85,B 0,C 180,E1 -23900.55,E2 -23900.55} C_VEL
LIN {X 0,Y 178.93,Z 682.686,A -85,B 0,C 180,E1 -23903.902,E2 -23903.902} C_VEL
LIN {X 0,Y 170.966,Z 683.104,A -85,B 0,C 180,E1 -23907.697,E2 -23907.697} C_VEL
LIN {X 0,Y 164.051,Z 682.525,A -85,B 0,C 180,E1 -23911.885,E2 -23911.885} C_VEL
LIN {X 0,Y 158.422,Z 681.008,A -85,B 0,C 180,E1 -23916.468,E2 -23916.468} C_VEL
LIN {X 0,Y 154.066,Z 678.519,A -85,B 0,C 180,E1 -23921.379,E2 -23921.379} C_VEL
LIN {X 0,Y 150.99,Z 674.919,A -85,B 0,C 180,E1 -23926.542,E2 -23926.542} C_VEL
LIN {X 0,Y 149.155,Z 670.148,A -85,B 0,C 180,E1 -23931.874,E2 -23931.874} C_VEL
LIN {X 0,Y 148.703,Z 665.77,A -85,B 0,C 180,E1 -23935.935,E2 -23935.935} C_VEL
LIN {X 0,Y 148.491,Z 660.47,A -85,B 0,C 180,E1 -23940,E2 -23940} C_VEL
LIN {X 0,Y 148.604,Z 652.984,A -85,B 0,C 180,E1 -23944.739,E2 -23944.739} C_VEL
LIN {X 0,Y 149.123,Z 645.048,A -85,B 0,C 180,E1 -23948.898,E2 -23948.898} C_VEL
LIN {X 0,Y 150.085,Z 634.36,A -85,B 0,C 180,E1 -23953.541,E2 -23953.541} C_VEL
LIN {X 0,Y 150.475,Z 631.285,A -85,B 0,C 180,E1 -23954.972,E2 -23954.972} C_VEL
LIN {X 0,Y 150.63,Z 630.904,A -85,B 0,C 180,E1 -23955.562,E2 -23955.562} C_VEL
LIN {X 0,Y 150.989,Z 630.963,A -85,B 0,C 180,E1 -23956.217,E2 -23956.217} C_VEL
LIN {X 0,Y 159.315,Z 626.84,A -85,B 0,C 180,E1 -23962.12,E2 -23962.12} C_VEL
LIN {X 0,Y 163.568,Z 624.007,A -85,B 0,C 180,E1 -23964.091,E2 -23964.091} C_VEL
LIN {X 0,Y 165.42,Z 623.267,A -85,B 0,C 180,E1 -23965.142,E2 -23965.142} C_VEL
LIN {X 0,Y 168.374,Z 621.611,A -85,B 0,C 180,E1 -23966.492,E2 -23966.492} C_VEL
LIN {X 0,Y 172.574,Z 618.471,A -85,B 0,C 180,E1 -23967.926,E2 -23967.926} C_VEL
LIN {X 0,Y 174.719,Z 617.457,A -85,B 0,C 180,E1 -23968.862,E2 -23968.862} C_VEL
LIN {X 0,Y 177.295,Z 615.932,A -85,B 0,C 180,E1 -23969.834,E2 -23969.834} C_VEL
LIN {X 0,Y 181.114,Z 612.914,A -85,B 0,C 180,E1 -23970.941,E2 -23970.941} C_VEL
LIN {X 0,Y 185.57,Z 608.718,A -85,B 0,C 180,E1 -23972.02,E2 -23972.02} C_VEL
LIN {X 0,Y 188.815,Z 606.631,A -85,B 0,C 180,E1 -23973.035,E2 -23973.035} C_VEL
LIN {X 0,Y 192.202,Z 603.827,A -85,B 0,C 180,E1 -23973.892,E2 -23973.892} C_VEL
LIN {X 0,Y 197.159,Z 598.598,A -85,B 0,C 180,E1 -23974.928,E2 -23974.928} C_VEL
LIN {X 0,Y 203.371,Z 590.459,A -85,B 0,C 180,E1 -23975.979,E2 -23975.979} C_VEL
LIN {X 0,Y 206.838,Z 586.838,A -85,B 0,C 180,E1 -23976.762,E2 -23976.762} C_VEL
LIN {X 0,Y 203.129,Z 601.948,A -85,B 0,C 180,E1 -23977.881,E2 -23977.881} C_VEL
LIN {X 0,Y 198.752,Z 615.978,A -85,B 0,C 180,E1 -23979.281,E2 -23979.281} C_VEL
LIN {X 0,Y 194.183,Z 628.452,A -85,B 0,C 180,E1 -23980.928,E2 -23980.928} C_VEL
LIN {X 0,Y 188.561,Z 641.154,A -85,B 0,C 180,E1 -23982.991,E2 -23982.991} C_VEL
LIN {X 0,Y 182.767,Z 652.796,A -85,B 0,C 180,E1 -23985.43,E2 -23985.43} C_VEL
LIN {X 0,Y 176.81,Z 663.464,A -85,B 0,C 180,E1 -23988.256,E2 -23988.256} C_VEL
LIN {X 0,Y 170.479,Z 673.846,A -85,B 0,C 180,E1 -23991.802,E2 -23991.802} C_VEL
LIN {X 0,Y 165.726,Z 681.371,A -85,B 0,C 180,E1 -23995.075,E2 -23995.075} C_VEL
LIN {X 0,Y 161.293,Z 687.73,A -85,B 0,C 180,E1 -23998.474,E2 -23998.474} C_VEL
LIN {X 0,Y 156.378,Z 694.763,A -85,B 0,C 180,E1 -24003.293,E2 -24003.293} C_VEL
LIN {X 0,Y 152.613,Z 700.295,A -85,B 0,C 180,E1 -24008.382,E2 -24008.382} C_VEL
LIN {X 0,Y 149.868,Z 704.479,A -85,B 0,C 180,E1 -24013.658,E2 -24013.658} C_VEL
LIN {X 0,Y 148.276,Z 707.418,A -85,B 0,C 180,E1 -24019.071,E2 -24019.071} C_VEL
LIN {X 0,Y 147.612,Z 709.177,A -85,B 0,C 180,E1 -24024.535,E2 -24024.535} C_VEL
LIN {X 0,Y 147.589,Z 709.784,A -85,B 0,C 180,E1 -24030,E2 -24030} C_VEL
LIN {X 0,Y 147.611,Z 709.205,A -85,B 0,C 180,E1 -24035.464,E2 -24035.464} C_VEL
LIN {X 0,Y 148.273,Z 707.484,A -85,B 0,C 180,E1 -24040.929,E2 -24040.929} C_VEL
LIN {X 0,Y 149.845,Z 704.59,A -85,B 0,C 180,E1 -24046.344,E2 -24046.344} C_VEL
LIN {X 0,Y 152.564,Z 700.455,A -85,B 0,C 180,E1 -24051.624,E2 -24051.624} C_VEL
LIN {X 0,Y 156.34,Z 694.966,A -85,B 0,C 180,E1 -24056.713,E2 -24056.713} C_VEL
LIN {X 0,Y 161.211,Z 687.975,A -85,B 0,C 180,E1 -24061.543,E2 -24061.543} C_VEL
LIN {X 0,Y 166.41,Z 680.489,A -85,B 0,C 180,E1 -24065.5,E2 -24065.5} C_VEL
LIN {X 0,Y 172.141,Z 671.423,A -85,B 0,C 180,E1 -24069.281,E2 -24069.281} C_VEL
LIN {X 0,Y 177.679,Z 662.255,A -85,B 0,C 180,E1 -24072.254,E2 -24072.254} C_VEL
LIN {X 0,Y 184.176,Z 650.382,A -85,B 0,C 180,E1 -24075.293,E2 -24075.293} C_VEL
LIN {X 0,Y 190.154,Z 638.263,A -85,B 0,C 180,E1 -24077.662,E2 -24077.662} C_VEL
LIN {X 0,Y 195.652,Z 625.074,A -85,B 0,C 180,E1 -24079.716,E2 -24079.716} C_VEL
LIN {X 0,Y 200.348,Z 611.844,A -85,B 0,C 180,E1 -24081.307,E2 -24081.307} C_VEL
LIN {X 0,Y 204.549,Z 597.543,A -85,B 0,C 180,E1 -24082.612,E2 -24082.612} C_VEL
LIN {X 0,Y 207.982,Z 582.78,A -85,B 0,C 180,E1 -24083.577,E2 -24083.577} C_VEL
LIN {X 0,Y 210.436,Z 567.534,A -85,B 0,C 180,E1 -24084.289,E2 -24084.289} C_VEL
LIN {X 0,Y 212.74,Z 541.508,A -85,B 0,C 180,E1 -24085.054,E2 -24085.054} C_VEL
LIN {X 0,Y 217.368,Z 482.852,A -85,B 0,C 180,E1 -24086.657,E2 -24086.657} C_VEL
LIN {X 0,Y 213.749,Z 473.938,A -85,B 0,C 180,E1 -24088.712,E2 -24088.712} C_VEL
LIN {X 0,Y 209.364,Z 464.37,A -85,B 0,C 180,E1 -24091.396,E2 -24091.396} C_VEL
LIN {X 0,Y 205.138,Z 456.21,A -85,B 0,C 180,E1 -24094.26,E2 -24094.26} C_VEL
LIN {X 0,Y 200.731,Z 448.449,A -85,B 0,C 180,E1 -24097.687,E2 -24097.687} C_VEL
LIN {X 0,Y 197.993,Z 443.888,A -85,B 0,C 180,E1 -24100.157,E2 -24100.157} C_VEL
LIN {X 0,Y 195.058,Z 439.262,A -85,B 0,C 180,E1 -24103.247,E2 -24103.247} C_VEL
LIN {X 0,Y 192.26,Z 434.925,A -85,B 0,C 180,E1 -24106.927,E2 -24106.927} C_VEL
LIN {X 0,Y 189.788,Z 431.185,A -85,B 0,C 180,E1 -24111.482,E2 -24111.482} C_VEL
LIN {X 0,Y 188.053,Z 427.983,A -85,B 0,C 180,E1 -24118.929,E2 -24118.929} C_VEL
LIN {X 0,Y 188.06,Z 427.763,A -85,B 0,C 180,E1 -24121.07,E2 -24121.07} C_VEL
LIN {X 0,Y 188.996,Z 429.687,A -85,B 0,C 180,E1 -24126.606,E2 -24126.606} C_VEL
LIN {X 0,Y 191.833,Z 433.344,A -85,B 0,C 180,E1 -24132.564,E2 -24132.564} C_VEL
LIN {X 0,Y 195.052,Z 437.9,A -85,B 0,C 180,E1 -24136.889,E2 -24136.889} C_VEL
LIN {X 0,Y 198.099,Z 442.371,A -85,B 0,C 180,E1 -24140.078,E2 -24140.078} C_VEL
LIN {X 0,Y 200.887,Z 446.678,A -85,B 0,C 180,E1 -24142.565,E2 -24142.565} C_VEL
LIN {X 0,Y 203.177,Z 450.293,A -85,B 0,C 180,E1 -24144.388,E2 -24144.388} C_VEL
LIN {X 0,Y 206.306,Z 455.303,A -85,B 0,C 180,E1 -24146.636,E2 -24146.636} C_VEL
LIN {X 0,Y 210.349,Z 462.276,A -85,B 0,C 180,E1 -24149.251,E2 -24149.251} C_VEL
LIN {X 0,Y 215.235,Z 471.686,A -85,B 0,C 180,E1 -24152.094,E2 -24152.094} C_VEL
LIN {X 0,Y 216.797,Z 475.119,A -85,B 0,C 180,E1 -24152.956,E2 -24152.956} C_VEL
LIN {X 0,Y 217.416,Z 477.237,A -85,B 0,C 180,E1 -24153.334,E2 -24153.334} C_VEL
LIN {X 0,Y 212.089,Z 545.36,A -85,B 0,C 180,E1 -24155.209,E2 -24155.209} C_VEL
LIN {X 0,Y 211.228,Z 551.222,A -85,B 0,C 180,E1 -24155.211,E2 -24155.211} C_VEL
LIN {X 0,Y 205.922,Z 570.171,A -85,B 0,C 180,E1 -24154.474,E2 -24154.474} C_VEL
LIN {X 0,Y 204.722,Z 575.91,A -85,B 0,C 180,E1 -24154.613,E2 -24154.613} C_VEL
LIN {X 0,Y 201.64,Z 590.783,A -85,B 0,C 180,E1 -24155.441,E2 -24155.441} C_VEL
LIN {X 0,Y 197.854,Z 604.659,A -85,B 0,C 180,E1 -24156.519,E2 -24156.519} C_VEL
LIN {X 0,Y 193.487,Z 617.824,A -85,B 0,C 180,E1 -24157.898,E2 -24157.898} C_VEL
LIN {X 0,Y 188.336,Z 630.875,A -85,B 0,C 180,E1 -24159.678,E2 -24159.678} C_VEL
LIN {X 0,Y 182.066,Z 644.221,A -85,B 0,C 180,E1 -24162.006,E2 -24162.006} C_VEL
LIN {X 0,Y 176.589,Z 654.36,A -85,B 0,C 180,E1 -24164.244,E2 -24164.244} C_VEL
LIN {X 0,Y 170.472,Z 664.702,A -85,B 0,C 180,E1 -24167.138,E2 -24167.138} C_VEL
LIN {X 0,Y 164.769,Z 673.465,A -85,B 0,C 180,E1 -24170.223,E2 -24170.223} C_VEL
LIN {X 0,Y 159.837,Z 680.967,A -85,B 0,C 180,E1 -24173.588,E2 -24173.588} C_VEL
LIN {X 0,Y 155.179,Z 687.322,A -85,B 0,C 180,E1 -24177.08,E2 -24177.08} C_VEL
LIN {X 0,Y 149.966,Z 694.341,A -85,B 0,C 180,E1 -24182.054,E2 -24182.054} C_VEL
LIN {X 0,Y 145.92,Z 699.852,A -85,B 0,C 180,E1 -24187.338,E2 -24187.338} C_VEL
LIN {X 0,Y 142.989,Z 704.005,A -85,B 0,C 180,E1 -24192.849,E2 -24192.849} C_VEL
LIN {X 0,Y 141.286,Z 706.911,A -85,B 0,C 180,E1 -24198.524,E2 -24198.524} C_VEL
LIN {X 0,Y 140.543,Z 708.642,A -85,B 0,C 180,E1 -24204.26,E2 -24204.26} C_VEL
LIN {X 0,Y 140.501,Z 709.229,A -85,B 0,C 180,E1 -24210,E2 -24210} C_VEL
LIN {X 0,Y 140.485,Z 709.074,A -85,B 0,C 180,E1 -24212.868,E2 -24212.868} C_VEL
LIN {X 0,Y 140.772,Z 707.899,A -85,B 0,C 180,E1 -24218.614,E2 -24218.614} C_VEL
LIN {X 0,Y 142.005,Z 705.566,A -85,B 0,C 180,E1 -24224.327,E2 -24224.327} C_VEL
LIN {X 0,Y 144.37,Z 702.02,A -85,B 0,C 180,E1 -24229.924,E2 -24229.924} C_VEL
LIN {X 0,Y 147.755,Z 697.179,A -85,B 0,C 180,E1 -24235.347,E2 -24235.347} C_VEL
LIN {X 0,Y 152.517,Z 690.908,A -85,B 0,C 180,E1 -24240.457,E2 -24240.457} C_VEL
LIN {X 0,Y 155.181,Z 687.802,A -85,B 0,C 180,E1 -24242.631,E2 -24242.631} C_VEL
LIN {X 0,Y 162.317,Z 687.277,A -85,B 0,C 180,E1 -24247.314,E2 -24247.314} C_VEL
LIN {X 0,Y 170.337,Z 686.067,A -85,B 0,C 180,E1 -24251.312,E2 -24251.312} C_VEL
LIN {X 0,Y 179.409,Z 684.09,A -85,B 0,C 180,E1 -24254.839,E2 -24254.839} C_VEL
LIN {X 0,Y 184.347,Z 682.855,A -85,B 0,C 180,E1 -24256.415,E2 -24256.415} C_VEL
LIN {X 0,Y 187.699,Z 681.846,A -85,B 0,C 180,E1 -24257.626,E2 -24257.626} C_VEL
LIN {X 0,Y 177.9,Z 683.247,A -85,B 0,C 180,E1 -24260.796,E2 -24260.796} C_VEL
LIN {X 0,Y 169.035,Z 683.71,A -85,B 0,C 180,E1 -24264.403,E2 -24264.403} C_VEL
LIN {X 0,Y 161.318,Z 683.233,A -85,B 0,C 180,E1 -24268.481,E2 -24268.481} C_VEL
LIN {X 0,Y 154.691,Z 681.863,A -85,B 0,C 180,E1 -24272.979,E2 -24272.979} C_VEL
LIN {X 0,Y 149.501,Z 679.497,A -85,B 0,C 180,E1 -24277.909,E2 -24277.909} C_VEL
LIN {X 0,Y 144.808,Z 675.13,A -85,B 0,C 180,E1 -24284.518,E2 -24284.518} C_VEL
LIN {X 0,Y 142.376,Z 669.596,A -85,B 0,C 180,E1 -24290.841,E2 -24290.841} C_VEL
LIN {X 0,Y 141.776,Z 664.31,A -85,B 0,C 180,E1 -24295.736,E2 -24295.736} C_VEL
LIN {X 0,Y 141.548,Z 657.705,A -85,B 0,C 180,E1 -24300.712,E2 -24300.712} C_VEL
LIN {X 0,Y 141.757,Z 649.614,A -85,B 0,C 180,E1 -24305.691,E2 -24305.691} C_VEL
LIN {X 0,Y 142.361,Z 640.583,A -85,B 0,C 180,E1 -24310.309,E2 -24310.309} C_VEL
LIN {X 0,Y 142.427,Z 639.103,A -85,B 0,C 180,E1 -24311.384,E2 -24311.384} C_VEL
LIN {X 0,Y 142.926,Z 638.963,A -85,B 0,C 180,E1 -24312.784,E2 -24312.784} C_VEL
LIN {X 0,Y 144.086,Z 638.467,A -85,B 0,C 180,E1 -24314.116,E2 -24314.116} C_VEL
LIN {X 0,Y 145.846,Z 637.331,A -85,B 0,C 180,E1 -24315.471,E2 -24315.471} C_VEL
LIN {X 0,Y 153.646,Z 633.924,A -85,B 0,C 180,E1 -24321.465,E2 -24321.465} C_VEL
LIN {X 0,Y 157.478,Z 632.169,A -85,B 0,C 180,E1 -24323.682,E2 -24323.682} C_VEL
LIN {X 0,Y 161.99,Z 629.488,A -85,B 0,C 180,E1 -24325.713,E2 -24325.713} C_VEL
LIN {X 0,Y 166.322,Z 627.415,A -85,B 0,C 180,E1 -24327.698,E2 -24327.698} C_VEL
LIN {X 0,Y 171.548,Z 623.95,A -85,B 0,C 180,E1 -24329.447,E2 -24329.447} C_VEL
LIN {X 0,Y 176.301,Z 621.51,A -85,B 0,C 180,E1 -24331.214,E2 -24331.214} C_VEL
LIN {X 0,Y 180.548,Z 618.469,A -85,B 0,C 180,E1 -24332.36,E2 -24332.36} C_VEL
LIN {X 0,Y 185.222,Z 614.37,A -85,B 0,C 180,E1 -24333.409,E2 -24333.409} C_VEL
LIN {X 0,Y 190.637,Z 610.727,A -85,B 0,C 180,E1 -24334.85,E2 -24334.85} C_VEL
LIN {X 0,Y 195.949,Z 605.992,A -85,B 0,C 180,E1 -24335.962,E2 -24335.962} C_VEL
LIN {X 0,Y 198.004,Z 603.892,A -85,B 0,C 180,E1 -24336.32,E2 -24336.32} C_VEL
LIN {X 0,Y 197.928,Z 605.096,A -85,B 0,C 180,E1 -24336.545,E2 -24336.545} C_VEL
LIN {X 0,Y 193.167,Z 619.226,A -85,B 0,C 180,E1 -24338.043,E2 -24338.043} C_VEL
LIN {X 0,Y 187.849,Z 632.544,A -85,B 0,C 180,E1 -24339.917,E2 -24339.917} C_VEL
LIN {X 0,Y 181.553,Z 645.631,A -85,B 0,C 180,E1 -24342.239,E2 -24342.239} C_VEL
LIN {X 0,Y 175.645,Z 656.582,A -85,B 0,C 180,E1 -24344.746,E2 -24344.746} C_VEL
LIN {X 0,Y 169.588,Z 666.661,A -85,B 0,C 180,E1 -24347.668,E2 -24347.668} C_VEL
LIN {X 0,Y 164.08,Z 675.17,A -85,B 0,C 180,E1 -24350.818,E2 -24350.818} C_VEL
LIN {X 0,Y 159.083,Z 682.462,A -85,B 0,C 180,E1 -24354.171,E2 -24354.171} C_VEL
LIN {X 0,Y 153.828,Z 689.641,A -85,B 0,C 180,E1 -24358.304,E2 -24358.304} C_VEL
LIN {X 0,Y 148.903,Z 696.282,A -85,B 0,C 180,E1 -24363.361,E2 -24363.361} C_VEL
LIN {X 0,Y 145.175,Z 701.477,A -85,B 0,C 180,E1 -24368.71,E2 -24368.71} C_VEL
LIN {X 0,Y 143.02,Z 704.466,A -85,B 0,C 180,E1 -24372.852,E2 -24372.852} C_VEL
LIN {X 0,Y 141.292,Z 707.404,A -85,B 0,C 180,E1 -24378.523,E2 -24378.523} C_VEL
LIN {X 0,Y 140.533,Z 709.163,A -85,B 0,C 180,E1 -24384.259,E2 -24384.259} C_VEL
LIN {X 0,Y 140.486,Z 709.77,A -85,B 0,C 180,E1 -24390,E2 -24390} C_VEL
LIN {X 0,Y 140.533,Z 709.191,A -85,B 0,C 180,E1 -24395.74,E2 -24395.74} C_VEL
LIN {X 0,Y 141.289,Z 707.47,A -85,B 0,C 180,E1 -24401.476,E2 -24401.476} C_VEL
LIN {X 0,Y 142.996,Z 704.575,A -85,B 0,C 180,E1 -24407.151,E2 -24407.151} C_VEL
LIN {X 0,Y 145.936,Z 700.439,A -85,B 0,C 180,E1 -24412.66,E2 -24412.66} C_VEL
LIN {X 0,Y 149.97,Z 694.949,A -85,B 0,C 180,E1 -24417.945,E2 -24417.945} C_VEL
LIN {X 0,Y 155.151,Z 687.957,A -85,B 0,C 180,E1 -24422.927,E2 -24422.927} C_VEL
LIN {X 0,Y 160.649,Z 680.47,A -85,B 0,C 180,E1 -24426.979,E2 -24426.979} C_VEL
LIN {X 0,Y 166.645,Z 671.451,A -85,B 0,C 180,E1 -24430.818,E2 -24430.818} C_VEL
LIN {X 0,Y 172.459,Z 662.233,A -85,B 0,C 180,E1 -24433.85,E2 -24433.85} C_VEL
LIN {X 0,Y 179.24,Z 650.357,A -85,B 0,C 180,E1 -24436.91,E2 -24436.91} C_VEL
LIN {X 0,Y 185.434,Z 638.235,A -85,B 0,C 180,E1 -24439.288,E2 -24439.288} C_VEL
LIN {X 0,Y 191.184,Z 624.89,A -85,B 0,C 180,E1 -24441.365,E2 -24441.365} C_VEL
LIN {X 0,Y 195.992,Z 611.806,A -85,B 0,C 180,E1 -24442.925,E2 -24442.925} C_VEL
LIN {X 0,Y 200.319,Z 597.496,A -85,B 0,C 180,E1 -24444.225,E2 -24444.225} C_VEL
LIN {X 0,Y 203.697,Z 583.453,A -85,B 0,C 180,E1 -24445.135,E2 -24445.135} C_VEL
LIN {X 0,Y 206.172,Z 568.806,A -85,B 0,C 180,E1 -24445.834,E2 -24445.834} C_VEL
LIN {X 0,Y 208.076,Z 549.657,A -85,B 0,C 180,E1 -24446.426,E2 -24446.426} C_VEL
LIN {X 0,Y 213.332,Z 485.745,A -85,B 0,C 180,E1 -24448.152,E2 -24448.152} C_VEL
LIN {X 0,Y 210.183,Z 477.861,A -85,B 0,C 180,E1 -24450.077,E2 -24450.077} C_VEL
LIN {X 0,Y 206.319,Z 469.149,A -85,B 0,C 180,E1 -24452.622,E2 -24452.622} C_VEL
LIN {X 0,Y 202.568,Z 461.618,A -85,B 0,C 180,E1 -24455.348,E2 -24455.348} C_VEL
LIN {X 0,Y 198.378,Z 453.996,A -85,B 0,C 180,E1 -24458.843,E2 -24458.843} C_VEL
LIN {X 0,Y 196.1,Z 450.075,A -85,B 0,C 180,E1 -24461.047,E2 -24461.047} C_VEL
LIN {X 0,Y 193.428,Z 445.677,A -85,B 0,C 180,E1 -24464.051,E2 -24464.051} C_VEL
LIN {X 0,Y 191.051,Z 441.779,A -85,B 0,C 180,E1 -24467.375,E2 -24467.375} C_VEL
LIN {X 0,Y 188.832,Z 438.245,A -85,B 0,C 180,E1 -24471.64,E2 -24471.64} C_VEL
LIN {X 0,Y 187.183,Z 435.067,A -85,B 0,C 180,E1 -24478.924,E2 -24478.924} C_VEL
LIN {X 0,Y 187.194,Z 434.819,A -85,B 0,C 180,E1 -24481.075,E2 -24481.075} C_VEL
LIN {X 0,Y 188.064,Z 436.724,A -85,B 0,C 180,E1 -24486.437,E2 -24486.437} C_VEL
LIN {X 0,Y 190.644,Z 440.172,A -85,B 0,C 180,E1 -24492.103,E2 -24492.103} C_VEL
LIN {X 0,Y 193.641,Z 444.608,A -85,B 0,C 180,E1 -24496.336,E2 -24496.336} C_VEL
LIN {X 0,Y 196.448,Z 448.914,A -85,B 0,C 180,E1 -24499.426,E2 -24499.426} C_VEL
LIN {X 0,Y 200.147,Z 454.711,A -85,B 0,C 180,E1 -24502.79,E2 -24502.79} C_VEL
LIN {X 0,Y 205.143,Z 463.153,A -85,B 0,C 180,E1 -24506.588,E2 -24506.588} C_VEL
LIN {X 0,Y 210.291,Z 472.942,A -85,B 0,C 180,E1 -24509.948,E2 -24509.948} C_VEL
LIN {X 0,Y 213.405,Z 479.603,A -85,B 0,C 180,E1 -24511.798,E2 -24511.798} C_VEL
LIN {X 0,Y 206.4,Z 564.161,A -85,B 0,C 180,E1 -24514.143,E2 -24514.143} C_VEL
LIN {X 0,Y 204.722,Z 575.91,A -85,B 0,C 180,E1 -24514.613,E2 -24514.613} C_VEL
LIN {X 0,Y 203.896,Z 579.725,A -85,B 0,C 180,E1 -24514.743,E2 -24514.743} C_VEL
LIN {X 0,Y 201.296,Z 587.199,A -85,B 0,C 180,E1 -24514.731,E2 -24514.731} C_VEL
LIN {X 0,Y 195.598,Z 599.882,A -85,B 0,C 180,E1 -24514.587,E2 -24514.587} C_VEL
LIN {X 0,Y 193.524,Z 605.313,A -85,B 0,C 180,E1 -24514.894,E2 -24514.894} C_VEL
LIN {X 0,Y 189.199,Z 617.859,A -85,B 0,C 180,E1 -24516.197,E2 -24516.197} C_VEL
LIN {X 0,Y 183.819,Z 631.038,A -85,B 0,C 180,E1 -24517.992,E2 -24517.992} C_VEL
LIN {X 0,Y 177.382,Z 644.247,A -85,B 0,C 180,E1 -24520.298,E2 -24520.298} C_VEL
LIN {X 0,Y 171.698,Z 654.383,A -85,B 0,C 180,E1 -24522.542,E2 -24522.542} C_VEL
LIN {X 0,Y 165.329,Z 664.724,A -85,B 0,C 180,E1 -24525.461,E2 -24525.461} C_VEL
LIN {X 0,Y 158.545,Z 674.678,A -85,B 0,C 180,E1 -24529.075,E2 -24529.075} C_VEL
LIN {X 0,Y 153.285,Z 682.093,A -85,B 0,C 180,E1 -24532.591,E2 -24532.591} C_VEL
LIN {X 0,Y 147.726,Z 689.251,A -85,B 0,C 180,E1 -24536.832,E2 -24536.832} C_VEL
LIN {X 0,Y 142.459,Z 695.876,A -85,B 0,C 180,E1 -24542.052,E2 -24542.052} C_VEL
LIN {X 0,Y 138.454,Z 701.049,A -85,B 0,C 180,E1 -24547.623,E2 -24547.623} C_VEL
LIN {X 0,Y 136.178,Z 704.02,A -85,B 0,C 180,E1 -24551.962,E2 -24551.962} C_VEL
LIN {X 0,Y 134.292,Z 706.925,A -85,B 0,C 180,E1 -24557.917,E2 -24557.917} C_VEL
LIN {X 0,Y 133.456,Z 708.656,A -85,B 0,C 180,E1 -24563.955,E2 -24563.955} C_VEL
LIN {X 0,Y 133.396,Z 709.092,A -85,B 0,C 180,E1 -24566.98,E2 -24566.98} C_VEL
LIN {X 0,Y 133.417,Z 709.242,A -85,B 0,C 180,E1 -24570,E2 -24570} C_VEL
LIN {X 0,Y 133.396,Z 709.088,A -85,B 0,C 180,E1 -24573.02,E2 -24573.02} C_VEL
LIN {X 0,Y 133.728,Z 707.912,A -85,B 0,C 180,E1 -24579.072,E2 -24579.072} C_VEL
LIN {X 0,Y 135.096,Z 705.579,A -85,B 0,C 180,E1 -24585.077,E2 -24585.077} C_VEL
LIN {X 0,Y 137.672,Z 702.034,A -85,B 0,C 180,E1 -24590.937,E2 -24590.937} C_VEL
LIN {X 0,Y 141.33,Z 697.193,A -85,B 0,C 180,E1 -24596.587,E2 -24596.587} C_VEL
LIN {X 0,Y 146.425,Z 690.922,A -85,B 0,C 180,E1 -24601.869,E2 -24601.869} C_VEL
LIN {X 0,Y 149.863,Z 687.098,A -85,B 0,C 180,E1 -24604.552,E2 -24604.552} C_VEL
LIN {X 0,Y 156.719,Z 686.916,A -85,B 0,C 180,E1 -24608.89,E2 -24608.89} C_VEL
LIN {X 0,Y 165.071,Z 686.067,A -85,B 0,C 180,E1 -24612.939,E2 -24612.939} C_VEL
LIN {X 0,Y 174.46,Z 684.465,A -85,B 0,C 180,E1 -24616.479,E2 -24616.479} C_VEL
LIN {X 0,Y 177.466,Z 683.842,A -85,B 0,C 180,E1 -24617.683,E2 -24617.683} C_VEL
LIN {X 0,Y 167.755,Z 684.33,A -85,B 0,C 180,E1 -24621.067,E2 -24621.067} C_VEL
LIN {X 0,Y 159.175,Z 683.936,A -85,B 0,C 180,E1 -24624.972,E2 -24624.972} C_VEL
LIN {X 0,Y 151.701,Z 682.66,A -85,B 0,C 180,E1 -24629.363,E2 -24629.363} C_VEL
LIN {X 0,Y 145.555,Z 680.411,A -85,B 0,C 180,E1 -24634.243,E2 -24634.243} C_VEL
LIN {X 0,Y 140.736,Z 677.223,A -85,B 0,C 180,E1 -24639.54,E2 -24639.54} C_VEL
LIN {X 0,Y 137.373,Z 673.015,A -85,B 0,C 180,E1 -24645.179,E2 -24645.179} C_VEL
LIN {X 0,Y 135.362,Z 667.604,A -85,B 0,C 180,E1 -24651.039,E2 -24651.039} C_VEL
LIN {X 0,Y 134.864,Z 662.696,A -85,B 0,C 180,E1 -24655.517,E2 -24655.517} C_VEL
LIN {X 0,Y 134.636,Z 655.782,A -85,B 0,C 180,E1 -24660.748,E2 -24660.748} C_VEL
LIN {X 0,Y 134.866,Z 646.683,A -85,B 0,C 180,E1 -24666.542,E2 -24666.542} C_VEL
LIN {X 0,Y 134.845,Z 646.351,A -85,B 0,C 180,E1 -24667.545,E2 -24667.545} C_VEL
LIN {X 0,Y 135.358,Z 646.247,A -85,B 0,C 180,E1 -24668.961,E2 -24668.961} C_VEL
LIN {X 0,Y 137.843,Z 644.7,A -85,B 0,C 180,E1 -24671.768,E2 -24671.768} C_VEL
LIN {X 0,Y 139.825,Z 644.168,A -85,B 0,C 180,E1 -24674.556,E2 -24674.556} C_VEL
LIN {X 0,Y 143.023,Z 642.598,A -85,B 0,C 180,E1 -24677.148,E2 -24677.148} C_VEL
LIN {X 0,Y 149.702,Z 639.879,A -85,B 0,C 180,E1 -24682.06,E2 -24682.06} C_VEL
LIN {X 0,Y 155.392,Z 637.466,A -85,B 0,C 180,E1 -24685.236,E2 -24685.236} C_VEL
LIN {X 0,Y 160.42,Z 634.772,A -85,B 0,C 180,E1 -24687.388,E2 -24687.388} C_VEL
LIN {X 0,Y 164.979,Z 632.683,A -85,B 0,C 180,E1 -24689.283,E2 -24689.283} C_VEL
LIN {X 0,Y 170.483,Z 629.294,A -85,B 0,C 180,E1 -24691.018,E2 -24691.018} C_VEL
LIN {X 0,Y 175.314,Z 626.95,A -85,B 0,C 180,E1 -24692.663,E2 -24692.663} C_VEL
LIN {X 0,Y 181.515,Z 622.648,A -85,B 0,C 180,E1 -24694.184,E2 -24694.184} C_VEL
LIN {X 0,Y 184.665,Z 620.08,A -85,B 0,C 180,E1 -24694.811,E2 -24694.811} C_VEL
LIN {X 0,Y 189.687,Z 616.79,A -85,B 0,C 180,E1 -24696.028,E2 -24696.028} C_VEL
LIN {X 0,Y 184.559,Z 629.807,A -85,B 0,C 180,E1 -24697.799,E2 -24697.799} C_VEL
LIN {X 0,Y 178.58,Z 642.271,A -85,B 0,C 180,E1 -24699.877,E2 -24699.877} C_VEL
LIN {X 0,Y 172.899,Z 652.76,A -85,B 0,C 180,E1 -24702.112,E2 -24702.112} C_VEL
LIN {X 0,Y 166.436,Z 663.43,A -85,B 0,C 180,E1 -24704.984,E2 -24704.984} C_VEL
LIN {X 0,Y 159.47,Z 673.815,A -85,B 0,C 180,E1 -24708.618,E2 -24708.618} C_VEL
LIN {X 0,Y 153.368,Z 682.447,A -85,B 0,C 180,E1 -24712.614,E2 -24712.614} C_VEL
LIN {X 0,Y 147.796,Z 689.627,A -85,B 0,C 180,E1 -24716.848,E2 -24716.848} C_VEL
LIN {X 0,Y 142.539,Z 696.267,A -85,B 0,C 180,E1 -24722.069,E2 -24722.069} C_VEL
LIN {X 0,Y 138.515,Z 701.463,A -85,B 0,C 180,E1 -24727.633,E2 -24727.633} C_VEL
LIN {X 0,Y 136.211,Z 704.452,A -85,B 0,C 180,E1 -24731.966,E2 -24731.966} C_VEL
LIN {X 0,Y 134.298,Z 707.391,A -85,B 0,C 180,E1 -24737.917,E2 -24737.917} C_VEL
LIN {X 0,Y 133.45,Z 709.15,A -85,B 0,C 180,E1 -24743.954,E2 -24743.954} C_VEL
LIN {X 0,Y 133.392,Z 709.757,A -85,B 0,C 180,E1 -24750,E2 -24750} C_VEL
LIN {X 0,Y 133.45,Z 709.177,A -85,B 0,C 180,E1 -24756.046,E2 -24756.046} C_VEL
LIN {X 0,Y 134.294,Z 707.455,A -85,B 0,C 180,E1 -24762.083,E2 -24762.083} C_VEL
LIN {X 0,Y 136.186,Z 704.56,A -85,B 0,C 180,E1 -24768.037,E2 -24768.037} C_VEL
LIN {X 0,Y 139.361,Z 700.423,A -85,B 0,C 180,E1 -24773.793,E2 -24773.793} C_VEL
LIN {X 0,Y 142.46,Z 696.442,A -85,B 0,C 180,E1 -24777.947,E2 -24777.947} C_VEL
LIN {X 0,Y 147.714,Z 689.841,A -85,B 0,C 180,E1 -24783.171,E2 -24783.171} C_VEL
LIN {X 0,Y 153.285,Z 682.713,A -85,B 0,C 180,E1 -24787.409,E2 -24787.409} C_VEL
LIN {X 0,Y 159.443,Z 674.019,A -85,B 0,C 180,E1 -24791.467,E2 -24791.467} C_VEL
LIN {X 0,Y 166.329,Z 663.82,A -85,B 0,C 180,E1 -24795.052,E2 -24795.052} C_VEL
LIN {X 0,Y 172.775,Z 653.229,A -85,B 0,C 180,E1 -24797.932,E2 -24797.932} C_VEL
LIN {X 0,Y 179.103,Z 641.682,A -85,B 0,C 180,E1 -24800.361,E2 -24800.361} C_VEL
LIN {X 0,Y 184.923,Z 629.345,A -85,B 0,C 180,E1 -24802.416,E2 -24802.416} C_VEL
LIN {X 0,Y 189.854,Z 617.127,A -85,B 0,C 180,E1 -24804.028,E2 -24804.028} C_VEL
LIN {X 0,Y 194.645,Z 602.939,A -85,B 0,C 180,E1 -24805.455,E2 -24805.455} C_VEL
LIN {X 0,Y 198.538,Z 588.533,A -85,B 0,C 180,E1 -24806.52,E2 -24806.52} C_VEL
LIN {X 0,Y 201.627,Z 573.194,A -85,B 0,C 180,E1 -24807.304,E2 -24807.304} C_VEL
LIN {X 0,Y 203.53,Z 558.078,A -85,B 0,C 180,E1 -24807.839,E2 -24807.839} C_VEL
LIN {X 0,Y 209.43,Z 488.589,A -85,B 0,C 180,E1 -24809.714,E2 -24809.714} C_VEL
LIN {X 0,Y 205.16,Z 477.907,A -85,B 0,C 180,E1 -24812.592,E2 -24812.592} C_VEL
LIN {X 0,Y 200.969,Z 468.787,A -85,B 0,C 180,E1 -24815.738,E2 -24815.738} C_VEL
LIN {X 0,Y 196.869,Z 460.947,A -85,B 0,C 180,E1 -24819.29,E2 -24819.29} C_VEL
LIN {X 0,Y 194.434,Z 456.508,A -85,B 0,C 180,E1 -24821.766,E2 -24821.766} C_VEL
LIN {X 0,Y 191.85,Z 452.075,A -85,B 0,C 180,E1 -24824.858,E2 -24824.858} C_VEL
LIN {X 0,Y 189.65,Z 448.316,A -85,B 0,C 180,E1 -24828.169,E2 -24828.169} C_VEL
LIN {X 0,Y 187.723,Z 445.045,A -85,B 0,C 180,E1 -24832.2,E2 -24832.2} C_VEL
LIN {X 0,Y 186.306,Z 441.973,A -85,B 0,C 180,E1 -24839.459,E2 -24839.459} C_VEL
LIN {X 0,Y 186.347,Z 442.02,A -85,B 0,C 180,E1 -24841.621,E2 -24841.621} C_VEL
LIN {X 0,Y 187.193,Z 443.869,A -85,B 0,C 180,E1 -24846.467,E2 -24846.467} C_VEL
LIN {X 0,Y 189.467,Z 447,A -85,B 0,C 180,E1 -24851.636,E2 -24851.636} C_VEL
LIN {X 0,Y 192.247,Z 451.322,A -85,B 0,C 180,E1 -24855.777,E2 -24855.777} C_VEL
LIN {X 0,Y 194.982,Z 455.7,A -85,B 0,C 180,E1 -24858.929,E2 -24858.929} C_VEL
LIN {X 0,Y 198.457,Z 461.498,A -85,B 0,C 180,E1 -24862.239,E2 -24862.239} C_VEL
LIN {X 0,Y 202.733,Z 468.93,A -85,B 0,C 180,E1 -24865.653,E2 -24865.653} C_VEL
LIN {X 0,Y 207.637,Z 478.652,A -85,B 0,C 180,E1 -24869.045,E2 -24869.045} C_VEL
LIN {X 0,Y 209.525,Z 482.748,A -85,B 0,C 180,E1 -24870.242,E2 -24870.242} C_VEL
LIN {X 0,Y 202.568,Z 563.725,A -85,B 0,C 180,E1 -24872.466,E2 -24872.466} C_VEL
LIN {X 0,Y 200.423,Z 577.905,A -85,B 0,C 180,E1 -24873.04,E2 -24873.04} C_VEL
LIN {X 0,Y 197.292,Z 592.106,A -85,B 0,C 180,E1 -24873.856,E2 -24873.856} C_VEL
LIN {X 0,Y 193.524,Z 605.313,A -85,B 0,C 180,E1 -24874.894,E2 -24874.894} C_VEL
LIN {X 0,Y 191.383,Z 610.765,A -85,B 0,C 180,E1 -24875.26,E2 -24875.26} C_VEL
LIN {X 0,Y 186.554,Z 619.375,A -85,B 0,C 180,E1 -24875.518,E2 -24875.518} C_VEL
LIN {X 0,Y 181.426,Z 627.713,A -85,B 0,C 180,E1 -24875.887,E2 -24875.887} C_VEL
LIN {X 0,Y 178.771,Z 632.64,A -85,B 0,C 180,E1 -24876.453,E2 -24876.453} C_VEL
LIN {X 0,Y 172.247,Z 645.331,A -85,B 0,C 180,E1 -24878.709,E2 -24878.709} C_VEL
LIN {X 0,Y 165.821,Z 656.268,A -85,B 0,C 180,E1 -24881.21,E2 -24881.21} C_VEL
LIN {X 0,Y 159.237,Z 666.347,A -85,B 0,C 180,E1 -24884.177,E2 -24884.177} C_VEL
LIN {X 0,Y 152.014,Z 676.432,A -85,B 0,C 180,E1 -24888.092,E2 -24888.092} C_VEL
LIN {X 0,Y 145.858,Z 684.326,A -85,B 0,C 180,E1 -24892.096,E2 -24892.096} C_VEL
LIN {X 0,Y 140.281,Z 691.065,A -85,B 0,C 180,E1 -24896.558,E2 -24896.558} C_VEL
LIN {X 0,Y 134.462,Z 697.935,A -85,B 0,C 180,E1 -24902.69,E2 -24902.69} C_VEL
LIN {X 0,Y 131,Z 702.121,A -85,B 0,C 180,E1 -24907.943,E2 -24907.943} C_VEL
LIN {X 0,Y 128.193,Z 705.638,A -85,B 0,C 180,E1 -24914.091,E2 -24914.091} C_VEL
LIN {X 0,Y 126.706,Z 707.949,A -85,B 0,C 180,E1 -24920.422,E2 -24920.422} C_VEL
LIN {X 0,Y 126.301,Z 709.106,A -85,B 0,C 180,E1 -24926.811,E2 -24926.811} C_VEL
LIN {X 0,Y 126.32,Z 709.256,A -85,B 0,C 180,E1 -24930,E2 -24930} C_VEL
LIN {X 0,Y 126.301,Z 709.102,A -85,B 0,C 180,E1 -24933.19,E2 -24933.19} C_VEL
LIN {X 0,Y 126.706,Z 707.926,A -85,B 0,C 180,E1 -24939.579,E2 -24939.579} C_VEL
LIN {X 0,Y 128.195,Z 705.593,A -85,B 0,C 180,E1 -24945.91,E2 -24945.91} C_VEL
LIN {X 0,Y 131.002,Z 702.047,A -85,B 0,C 180,E1 -24952.058,E2 -24952.058} C_VEL
LIN {X 0,Y 134.967,Z 697.207,A -85,B 0,C 180,E1 -24957.947,E2 -24957.947} C_VEL
LIN {X 0,Y 140.411,Z 690.936,A -85,B 0,C 180,E1 -24963.408,E2 -24963.408} C_VEL
LIN {X 0,Y 144.817,Z 686.299,A -85,B 0,C 180,E1 -24966.694,E2 -24966.694} C_VEL
LIN {X 0,Y 155.478,Z 686.212,A -85,B 0,C 180,E1 -24972.691,E2 -24972.691} C_VEL
LIN {X 0,Y 164.683,Z 685.38,A -85,B 0,C 180,E1 -24976.51,E2 -24976.51} C_VEL
LIN {X 0,Y 167.225,Z 684.956,A -85,B 0,C 180,E1 -24977.745,E2 -24977.745} C_VEL
LIN {X 0,Y 157.738,Z 684.629,A -85,B 0,C 180,E1 -24981.408,E2 -24981.408} C_VEL
LIN {X 0,Y 149.401,Z 683.398,A -85,B 0,C 180,E1 -24985.633,E2 -24985.633} C_VEL
LIN {X 0,Y 142.226,Z 681.27,A -85,B 0,C 180,E1 -24990.387,E2 -24990.387} C_VEL
LIN {X 0,Y 136.495,Z 678.262,A -85,B 0,C 180,E1 -24995.675,E2 -24995.675} C_VEL
LIN {X 0,Y 131.358,Z 673.035,A -85,B 0,C 180,E1 -25002.887,E2 -25002.887} C_VEL
LIN {X 0,Y 128.874,Z 667.627,A -85,B 0,C 180,E1 -25008.998,E2 -25008.998} C_VEL
LIN {X 0,Y 127.989,Z 660.933,A -85,B 0,C 180,E1 -25015.276,E2 -25015.276} C_VEL
LIN {X 0,Y 127.7,Z 653.747,A -85,B 0,C 180,E1 -25020.986,E2 -25020.986} C_VEL
LIN {X 0,Y 127.556,Z 653.444,A -85,B 0,C 180,E1 -25022.369,E2 -25022.369} C_VEL
LIN {X 0,Y 127.645,Z 653.435,A -85,B 0,C 180,E1 -25023.157,E2 -25023.157} C_VEL
LIN {X 0,Y 129.217,Z 652.321,A -85,B 0,C 180,E1 -25026.245,E2 -25026.245} C_VEL
LIN {X 0,Y 130.778,Z 651.634,A -85,B 0,C 180,E1 -25029.278,E2 -25029.278} C_VEL
LIN {X 0,Y 133.234,Z 650.361,A -85,B 0,C 180,E1 -25032.181,E2 -25032.181} C_VEL
LIN {X 0,Y 135.481,Z 649.698,A -85,B 0,C 180,E1 -25035.033,E2 -25035.033} C_VEL
LIN {X 0,Y 149.557,Z 644.129,A -85,B 0,C 180,E1 -25045.02,E2 -25045.02} C_VEL
LIN {X 0,Y 153.982,Z 642.203,A -85,B 0,C 180,E1 -25047.157,E2 -25047.157} C_VEL
LIN {X 0,Y 158.851,Z 639.902,A -85,B 0,C 180,E1 -25049.122,E2 -25049.122} C_VEL
LIN {X 0,Y 164.146,Z 637.519,A -85,B 0,C 180,E1 -25051.094,E2 -25051.094} C_VEL
LIN {X 0,Y 169.399,Z 634.521,A -85,B 0,C 180,E1 -25052.639,E2 -25052.639} C_VEL
LIN {X 0,Y 174.729,Z 632.019,A -85,B 0,C 180,E1 -25054.272,E2 -25054.272} C_VEL
LIN {X 0,Y 180.834,Z 628.041,A -85,B 0,C 180,E1 -25055.66,E2 -25055.66} C_VEL
LIN {X 0,Y 180.136,Z 630.12,A -85,B 0,C 180,E1 -25056.06,E2 -25056.06} C_VEL
LIN {X 0,Y 174.116,Z 642.252,A -85,B 0,C 180,E1 -25058.085,E2 -25058.085} C_VEL
LIN {X 0,Y 168.208,Z 652.742,A -85,B 0,C 180,E1 -25060.313,E2 -25060.313} C_VEL
LIN {X 0,Y 161.47,Z 663.414,A -85,B 0,C 180,E1 -25063.193,E2 -25063.193} C_VEL
LIN {X 0,Y 154.166,Z 673.8,A -85,B 0,C 180,E1 -25066.858,E2 -25066.858} C_VEL
LIN {X 0,Y 147.772,Z 682.432,A -85,B 0,C 180,E1 -25070.937,E2 -25070.937} C_VEL
LIN {X 0,Y 141.853,Z 689.612,A -85,B 0,C 180,E1 -25075.266,E2 -25075.266} C_VEL
LIN {X 0,Y 136.26,Z 696.253,A -85,B 0,C 180,E1 -25080.66,E2 -25080.66} C_VEL
LIN {X 0,Y 131.915,Z 701.45,A -85,B 0,C 180,E1 -25086.448,E2 -25086.448} C_VEL
LIN {X 0,Y 129.442,Z 704.439,A -85,B 0,C 180,E1 -25090.988,E2 -25090.988} C_VEL
LIN {X 0,Y 127.332,Z 707.377,A -85,B 0,C 180,E1 -25097.245,E2 -25097.245} C_VEL
LIN {X 0,Y 126.391,Z 709.136,A -85,B 0,C 180,E1 -25103.614,E2 -25103.614} C_VEL
LIN {X 0,Y 126.309,Z 709.743,A -85,B 0,C 180,E1 -25110,E2 -25110} C_VEL
LIN {X 0,Y 126.373,Z 709.163,A -85,B 0,C 180,E1 -25116.386,E2 -25116.386} C_VEL
LIN {X 0,Y 127.328,Z 707.441,A -85,B 0,C 180,E1 -25122.755,E2 -25122.755} C_VEL
LIN {X 0,Y 129.418,Z 704.546,A -85,B 0,C 180,E1 -25129.015,E2 -25129.015} C_VEL
LIN {X 0,Y 132.842,Z 700.408,A -85,B 0,C 180,E1 -25135.039,E2 -25135.039} C_VEL
LIN {X 0,Y 136.189,Z 696.426,A -85,B 0,C 180,E1 -25139.356,E2 -25139.356} C_VEL
LIN {X 0,Y 141.776,Z 689.824,A -85,B 0,C 180,E1 -25144.755,E2 -25144.755} C_VEL
LIN {X 0,Y 147.678,Z 682.695,A -85,B 0,C 180,E1 -25149.092,E2 -25149.092} C_VEL
LIN {X 0,Y 154.072,Z 674.122,A -85,B 0,C 180,E1 -25153.174,E2 -25153.174} C_VEL
LIN {X 0,Y 161.371,Z 663.799,A -85,B 0,C 180,E1 -25156.843,E2 -25156.843} C_VEL
LIN {X 0,Y 168.072,Z 653.205,A -85,B 0,C 180,E1 -25159.741,E2 -25159.741} C_VEL
LIN {X 0,Y 174.656,Z 641.654,A -85,B 0,C 180,E1 -25162.157,E2 -25162.157} C_VEL
LIN {X 0,Y 180.655,Z 629.313,A -85,B 0,C 180,E1 -25164.212,E2 -25164.212} C_VEL
LIN {X 0,Y 185.765,Z 617.089,A -85,B 0,C 180,E1 -25165.803,E2 -25165.803} C_VEL
LIN {X 0,Y 190.704,Z 602.892,A -85,B 0,C 180,E1 -25167.215,E2 -25167.215} C_VEL
LIN {X 0,Y 194.717,Z 588.472,A -85,B 0,C 180,E1 -25168.26,E2 -25168.26} C_VEL
LIN {X 0,Y 197.835,Z 573.412,A -85,B 0,C 180,E1 -25169.022,E2 -25169.022} C_VEL
LIN {X 0,Y 199.813,Z 558.209,A -85,B 0,C 180,E1 -25169.557,E2 -25169.557} C_VEL
LIN {X 0,Y 205.664,Z 491.468,A -85,B 0,C 180,E1 -25171.345,E2 -25171.345} C_VEL
LIN {X 0,Y 201.742,Z 481.532,A -85,B 0,C 180,E1 -25174.223,E2 -25174.223} C_VEL
LIN {X 0,Y 197.934,Z 473.064,A -85,B 0,C 180,E1 -25177.356,E2 -25177.356} C_VEL
LIN {X 0,Y 194.397,Z 465.99,A -85,B 0,C 180,E1 -25180.737,E2 -25180.737} C_VEL
LIN {X 0,Y 192.254,Z 462.006,A -85,B 0,C 180,E1 -25183.132,E2 -25183.132} C_VEL
LIN {X 0,Y 190.384,Z 458.609,A -85,B 0,C 180,E1 -25185.571,E2 -25185.571} C_VEL
LIN {X 0,Y 188.349,Z 454.945,A -85,B 0,C 180,E1 -25188.861,E2 -25188.861} C_VEL
LIN {X 0,Y 186.75,Z 452.053,A -85,B 0,C 180,E1 -25192.431,E2 -25192.431} C_VEL
LIN {X 0,Y 185.436,Z 449.055,A -85,B 0,C 180,E1 -25199.457,E2 -25199.457} C_VEL
LIN {X 0,Y 185.478,Z 449.101,A -85,B 0,C 180,E1 -25201.628,E2 -25201.628} C_VEL
LIN {X 0,Y 186.324,Z 450.987,A -85,B 0,C 180,E1 -25206.497,E2 -25206.497} C_VEL
LIN {X 0,Y 188.373,Z 453.945,A -85,B 0,C 180,E1 -25211.295,E2 -25211.295} C_VEL
LIN {X 0,Y 190.872,Z 458.041,A -85,B 0,C 180,E1 -25215.209,E2 -25215.209} C_VEL
LIN {X 0,Y 193.554,Z 462.532,A -85,B 0,C 180,E1 -25218.451,E2 -25218.451} C_VEL
LIN {X 0,Y 196.81,Z 468.355,A -85,B 0,C 180,E1 -25221.702,E2 -25221.702} C_VEL
LIN {X 0,Y 200.435,Z 474.872,A -85,B 0,C 180,E1 -25224.744,E2 -25224.744} C_VEL
LIN {X 0,Y 204.869,Z 484.03,A -85,B 0,C 180,E1 -25228.007,E2 -25228.007} C_VEL
LIN {X 0,Y 205.794,Z 486.092,A -85,B 0,C 180,E1 -25228.638,E2 -25228.638} C_VEL
LIN {X 0,Y 198.758,Z 564.688,A -85,B 0,C 180,E1 -25230.77,E2 -25230.77} C_VEL
LIN {X 0,Y 196.475,Z 578.866,A -85,B 0,C 180,E1 -25231.349,E2 -25231.349} C_VEL
LIN {X 0,Y 193.091,Z 593.43,A -85,B 0,C 180,E1 -25232.195,E2 -25232.195} C_VEL
LIN {X 0,Y 189.097,Z 606.693,A -85,B 0,C 180,E1 -25233.256,E2 -25233.256} C_VEL
LIN {X 0,Y 184.368,Z 619.617,A -85,B 0,C 180,E1 -25234.624,E2 -25234.624} C_VEL
LIN {X 0,Y 178.771,Z 632.64,A -85,B 0,C 180,E1 -25236.453,E2 -25236.453} C_VEL
LIN {X 0,Y 175.993,Z 637.54,A -85,B 0,C 180,E1 -25237.074,E2 -25237.074} C_VEL
LIN {X 0,Y 170.124,Z 645.247,A -85,B 0,C 180,E1 -25237.74,E2 -25237.74} C_VEL
LIN {X 0,Y 163.979,Z 652.63,A -85,B 0,C 180,E1 -25238.569,E2 -25238.569} C_VEL
LIN {X 0,Y 160.812,Z 656.899,A -85,B 0,C 180,E1 -25239.469,E2 -25239.469} C_VEL
LIN {X 0,Y 154.357,Z 666.368,A -85,B 0,C 180,E1 -25242.279,E2 -25242.279} C_VEL
LIN {X 0,Y 147.205,Z 675.791,A -85,B 0,C 180,E1 -25245.896,E2 -25245.896} C_VEL
LIN {X 0,Y 141.262,Z 683.237,A -85,B 0,C 180,E1 -25249.702,E2 -25249.702} C_VEL
LIN {X 0,Y 135.966,Z 689.285,A -85,B 0,C 180,E1 -25253.529,E2 -25253.529} C_VEL
LIN {X 0,Y 129.995,Z 695.909,A -85,B 0,C 180,E1 -25259.096,E2 -25259.096} C_VEL
LIN {X 0,Y 125.326,Z 701.079,A -85,B 0,C 180,E1 -25265.129,E2 -25265.129} C_VEL
LIN {X 0,Y 122.684,Z 704.049,A -85,B 0,C 180,E1 -25269.897,E2 -25269.897} C_VEL
LIN {X 0,Y 120.385,Z 706.954,A -85,B 0,C 180,E1 -25276.496,E2 -25276.496} C_VEL
LIN {X 0,Y 119.31,Z 708.684,A -85,B 0,C 180,E1 -25283.235,E2 -25283.235} C_VEL
LIN {X 0,Y 119.233,Z 709.27,A -85,B 0,C 180,E1 -25290,E2 -25290} C_VEL
LIN {X 0,Y 119.311,Z 708.67,A -85,B 0,C 180,E1 -25296.766,E2 -25296.766} C_VEL
LIN {X 0,Y 120.386,Z 706.92,A -85,B 0,C 180,E1 -25303.505,E2 -25303.505} C_VEL
LIN {X 0,Y 122.688,Z 703.99,A -85,B 0,C 180,E1 -25310.103,E2 -25310.103} C_VEL
LIN {X 0,Y 126.386,Z 699.809,A -85,B 0,C 180,E1 -25316.415,E2 -25316.415} C_VEL
LIN {X 0,Y 131.42,Z 694.278,A -85,B 0,C 180,E1 -25322.329,E2 -25322.329} C_VEL
LIN {X 0,Y 137.986,Z 687.254,A -85,B 0,C 180,E1 -25327.676,E2 -25327.676} C_VEL
LIN {X 0,Y 139.909,Z 685.431,A -85,B 0,C 180,E1 -25328.896,E2 -25328.896} C_VEL
LIN {X 0,Y 150.343,Z 685.698,A -85,B 0,C 180,E1 -25334.524,E2 -25334.524} C_VEL
LIN {X 0,Y 154.987,Z 685.501,A -85,B 0,C 180,E1 -25336.514,E2 -25336.514} C_VEL
LIN {X 0,Y 157.015,Z 685.31,A -85,B 0,C 180,E1 -25337.825,E2 -25337.825} C_VEL
LIN {X 0,Y 147.776,Z 684.115,A -85,B 0,C 180,E1 -25341.811,E2 -25341.811} C_VEL
LIN {X 0,Y 139.71,Z 682.087,A -85,B 0,C 180,E1 -25346.403,E2 -25346.403} C_VEL
LIN {X 0,Y 132.965,Z 679.185,A -85,B 0,C 180,E1 -25351.595,E2 -25351.595} C_VEL
LIN {X 0,Y 126.562,Z 674.203,A -85,B 0,C 180,E1 -25358.842,E2 -25358.842} C_VEL
LIN {X 0,Y 123.239,Z 669.018,A -85,B 0,C 180,E1 -25365.131,E2 -25365.131} C_VEL
LIN {X 0,Y 121.196,Z 661.012,A -85,B 0,C 180,E1 -25373.549,E2 -25373.549} C_VEL
LIN {X 0,Y 120.894,Z 660.354,A -85,B 0,C 180,E1 -25376.668,E2 -25376.668} C_VEL
LIN {X 0,Y 121.781,Z 659.263,A -85,B 0,C 180,E1 -25380,E2 -25380} C_VEL
LIN {X 0,Y 127.252,Z 656.276,A -85,B 0,C 180,E1 -25391.248,E2 -25391.248} C_VEL
LIN {X 0,Y 132.203,Z 654.51,A -85,B 0,C 180,E1 -25396.883,E2 -25396.883} C_VEL
LIN {X 0,Y 145.305,Z 649.796,A -85,B 0,C 180,E1 -25405.805,E2 -25405.805} C_VEL
LIN {X 0,Y 149.797,Z 648.047,A -85,B 0,C 180,E1 -25407.981,E2 -25407.981} C_VEL
LIN {X 0,Y 161.723,Z 643.007,A -85,B 0,C 180,E1 -25412.477,E2 -25412.477} C_VEL
LIN {X 0,Y 168.322,Z 639.604,A -85,B 0,C 180,E1 -25414.31,E2 -25414.31} C_VEL
LIN {X 0,Y 171.04,Z 638.466,A -85,B 0,C 180,E1 -25415.118,E2 -25415.118} C_VEL
LIN {X 0,Y 171.005,Z 640.078,A -85,B 0,C 180,E1 -25415.807,E2 -25415.807} C_VEL
LIN {X 0,Y 164.866,Z 650.797,A -85,B 0,C 180,E1 -25417.942,E2 -25417.942} C_VEL
LIN {X 0,Y 157.817,Z 661.788,A -85,B 0,C 180,E1 -25420.794,E2 -25420.794} C_VEL
LIN {X 0,Y 151.159,Z 671.039,A -85,B 0,C 180,E1 -25423.891,E2 -25423.891} C_VEL
LIN {X 0,Y 144.2,Z 680.128,A -85,B 0,C 180,E1 -25427.921,E2 -25427.921} C_VEL
LIN {X 0,Y 137.672,Z 687.673,A -85,B 0,C 180,E1 -25432.223,E2 -25432.223} C_VEL
LIN {X 0,Y 131.424,Z 694.708,A -85,B 0,C 180,E1 -25437.672,E2 -25437.672} C_VEL
LIN {X 0,Y 126.467,Z 700.24,A -85,B 0,C 180,E1 -25443.603,E2 -25443.603} C_VEL
LIN {X 0,Y 122.721,Z 704.425,A -85,B 0,C 180,E1 -25449.903,E2 -25449.903} C_VEL
LIN {X 0,Y 120.376,Z 707.364,A -85,B 0,C 180,E1 -25456.494,E2 -25456.494} C_VEL
LIN {X 0,Y 119.307,Z 709.122,A -85,B 0,C 180,E1 -25463.234,E2 -25463.234} C_VEL
LIN {X 0,Y 119.227,Z 709.729,A -85,B 0,C 180,E1 -25470,E2 -25470} C_VEL
LIN {X 0,Y 119.29,Z 709.149,A -85,B 0,C 180,E1 -25476.766,E2 -25476.766} C_VEL
LIN {X 0,Y 120.371,Z 707.426,A -85,B 0,C 180,E1 -25483.505,E2 -25483.505} C_VEL
LIN {X 0,Y 122.693,Z 704.531,A -85,B 0,C 180,E1 -25490.101,E2 -25490.101} C_VEL
LIN {X 0,Y 126.385,Z 700.392,A -85,B 0,C 180,E1 -25496.414,E2 -25496.414} C_VEL
LIN {X 0,Y 131.39,Z 694.9,A -85,B 0,C 180,E1 -25502.336,E2 -25502.336} C_VEL
LIN {X 0,Y 137.595,Z 687.905,A -85,B 0,C 180,E1 -25507.801,E2 -25507.801} C_VEL
LIN {X 0,Y 144.104,Z 680.414,A -85,B 0,C 180,E1 -25512.112,E2 -25512.112} C_VEL
LIN {X 0,Y 150.004,Z 672.763,A -85,B 0,C 180,E1 -25515.601,E2 -25515.601} C_VEL
LIN {X 0,Y 156.583,Z 663.777,A -85,B 0,C 180,E1 -25518.746,E2 -25518.746} C_VEL
LIN {X 0,Y 163.56,Z 653.18,A -85,B 0,C 180,E1 -25521.645,E2 -25521.645} C_VEL
LIN {X 0,Y 170.387,Z 641.626,A -85,B 0,C 180,E1 -25524.044,E2 -25524.044} C_VEL
LIN {X 0,Y 177.075,Z 628.2,A -85,B 0,C 180,E1 -25526.244,E2 -25526.244} C_VEL
LIN {X 0,Y 182.581,Z 615.149,A -85,B 0,C 180,E1 -25527.869,E2 -25527.869} C_VEL
LIN {X 0,Y 187.632,Z 600.649,A -85,B 0,C 180,E1 -25529.221,E2 -25529.221} C_VEL
LIN {X 0,Y 191.607,Z 586.205,A -85,B 0,C 180,E1 -25530.191,E2 -25530.191} C_VEL
LIN {X 0,Y 194.653,Z 571.009,A -85,B 0,C 180,E1 -25530.903,E2 -25530.903} C_VEL
LIN {X 0,Y 196.664,Z 554.27,A -85,B 0,C 180,E1 -25531.445,E2 -25531.445} C_VEL
LIN {X 0,Y 202.036,Z 494.531,A -85,B 0,C 180,E1 -25533.041,E2 -25533.041} C_VEL
LIN {X 0,Y 198.85,Z 486.085,A -85,B 0,C 180,E1 -25535.602,E2 -25535.602} C_VEL
LIN {X 0,Y 195.604,Z 478.514,A -85,B 0,C 180,E1 -25538.501,E2 -25538.501} C_VEL
LIN {X 0,Y 192.138,Z 471.233,A -85,B 0,C 180,E1 -25542.118,E2 -25542.118} C_VEL
LIN {X 0,Y 189.134,Z 465.448,A -85,B 0,C 180,E1 -25546.023,E2 -25546.023} C_VEL
LIN {X 0,Y 187.199,Z 461.791,A -85,B 0,C 180,E1 -25549.317,E2 -25549.317} C_VEL
LIN {X 0,Y 185.688,Z 458.899,A -85,B 0,C 180,E1 -25552.934,E2 -25552.934} C_VEL
LIN {X 0,Y 184.574,Z 455.97,A -85,B 0,C 180,E1 -25560,E2 -25560} C_VEL
LIN {X 0,Y 184.759,Z 456.679,A -85,B 0,C 180,E1 -25563.271,E2 -25563.271} C_VEL
LIN {X 0,Y 186.7,Z 459.937,A -85,B 0,C 180,E1 -25569.752,E2 -25569.752} C_VEL
LIN {X 0,Y 189.343,Z 464.403,A -85,B 0,C 180,E1 -25574.376,E2 -25574.376} C_VEL
LIN {X 0,Y 191.801,Z 468.779,A -85,B 0,C 180,E1 -25577.576,E2 -25577.576} C_VEL
LIN {X 0,Y 194.948,Z 474.669,A -85,B 0,C 180,E1 -25580.924,E2 -25580.924} C_VEL
LIN {X 0,Y 198.457,Z 481.324,A -85,B 0,C 180,E1 -25584.037,E2 -25584.037} C_VEL
LIN {X 0,Y 202.177,Z 489.375,A -85,B 0,C 180,E1 -25586.942,E2 -25586.942} C_VEL
LIN {X 0,Y 195.262,Z 564.524,A -85,B 0,C 180,E1 -25588.975,E2 -25588.975} C_VEL
LIN {X 0,Y 192.881,Z 578.938,A -85,B 0,C 180,E1 -25589.55,E2 -25589.55} C_VEL
LIN {X 0,Y 189.406,Z 593.483,A -85,B 0,C 180,E1 -25590.379,E2 -25590.379} C_VEL
LIN {X 0,Y 185.306,Z 606.735,A -85,B 0,C 180,E1 -25591.423,E2 -25591.423} C_VEL
LIN {X 0,Y 179.97,Z 620.75,A -85,B 0,C 180,E1 -25592.905,E2 -25592.905} C_VEL
LIN {X 0,Y 173.894,Z 634.179,A -85,B 0,C 180,E1 -25594.822,E2 -25594.822} C_VEL
LIN {X 0,Y 167.26,Z 646.414,A -85,B 0,C 180,E1 -25597.028,E2 -25597.028} C_VEL
LIN {X 0,Y 160.812,Z 656.899,A -85,B 0,C 180,E1 -25599.469,E2 -25599.469} C_VEL
LIN {X 0,Y 157.548,Z 661.141,A -85,B 0,C 180,E1 -25600.441,E2 -25600.441} C_VEL
LIN {X 0,Y 145.403,Z 672.625,A -85,B 0,C 180,E1 -25602.815,E2 -25602.815} C_VEL
LIN {X 0,Y 141.912,Z 676.17,A -85,B 0,C 180,E1 -25604.07,E2 -25604.07} C_VEL
LIN {X 0,Y 140.976,Z 677.274,A -85,B 0,C 180,E1 -25604.6,E2 -25604.6} C_VEL
LIN {X 0,Y 134.904,Z 684.362,A -85,B 0,C 180,E1 -25608.377,E2 -25608.377} C_VEL
LIN {X 0,Y 128.589,Z 691.099,A -85,B 0,C 180,E1 -25613.044,E2 -25613.044} C_VEL
LIN {X 0,Y 122.496,Z 697.339,A -85,B 0,C 180,E1 -25618.912,E2 -25618.912} C_VEL
LIN {X 0,Y 117.823,Z 702.151,A -85,B 0,C 180,E1 -25625.321,E2 -25625.321} C_VEL
LIN {X 0,Y 114.494,Z 705.667,A -85,B 0,C 180,E1 -25632.127,E2 -25632.127} C_VEL
LIN {X 0,Y 112.682,Z 707.977,A -85,B 0,C 180,E1 -25639.216,E2 -25639.216} C_VEL
LIN {X 0,Y 112.111,Z 709.134,A -85,B 0,C 180,E1 -25646.406,E2 -25646.406} C_VEL
LIN {X 0,Y 112.138,Z 709.283,A -85,B 0,C 180,E1 -25650,E2 -25650} C_VEL
LIN {X 0,Y 112.111,Z 709.129,A -85,B 0,C 180,E1 -25653.595,E2 -25653.595} C_VEL
LIN {X 0,Y 112.682,Z 707.953,A -85,B 0,C 180,E1 -25660.785,E2 -25660.785} C_VEL
LIN {X 0,Y 114.497,Z 705.62,A -85,B 0,C 180,E1 -25667.873,E2 -25667.873} C_VEL
LIN {X 0,Y 117.824,Z 702.074,A -85,B 0,C 180,E1 -25674.68,E2 -25674.68} C_VEL
LIN {X 0,Y 122.52,Z 697.234,A -85,B 0,C 180,E1 -25681.082,E2 -25681.082} C_VEL
LIN {X 0,Y 128.763,Z 690.973,A -85,B 0,C 180,E1 -25686.899,E2 -25686.899} C_VEL
LIN {X 0,Y 135.621,Z 684.384,A -85,B 0,C 180,E1 -25691.479,E2 -25691.479} C_VEL
LIN {X 0,Y 145.388,Z 684.953,A -85,B 0,C 180,E1 -25696.477,E2 -25696.477} C_VEL
LIN {X 0,Y 146.91,Z 684.806,A -85,B 0,C 180,E1 -25697.953,E2 -25697.953} C_VEL
LIN {X 0,Y 137.923,Z 682.853,A -85,B 0,C 180,E1 -25702.304,E2 -25702.304} C_VEL
LIN {X 0,Y 130.127,Z 680.016,A -85,B 0,C 180,E1 -25707.311,E2 -25707.311} C_VEL
LIN {X 0,Y 122.489,Z 675.23,A -85,B 0,C 180,E1 -25714.512,E2 -25714.512} C_VEL
LIN {X 0,Y 116.765,Z 668.377,A -85,B 0,C 180,E1 -25723.613,E2 -25723.613} C_VEL
LIN {X 0,Y 115.41,Z 667.832,A -85,B 0,C 180,E1 -25726.994,E2 -25726.994} C_VEL
LIN {X 0,Y 115.132,Z 667.18,A -85,B 0,C 180,E1 -25729.448,E2 -25729.448} C_VEL
LIN {X 0,Y 115.583,Z 665.838,A -85,B 0,C 180,E1 -25733.015,E2 -25733.015} C_VEL
LIN {X 0,Y 117.566,Z 663.51,A -85,B 0,C 180,E1 -25743.428,E2 -25743.428} C_VEL
LIN {X 0,Y 126.023,Z 660.103,A -85,B 0,C 180,E1 -25756.191,E2 -25756.191} C_VEL
LIN {X 0,Y 136.669,Z 656.6,A -85,B 0,C 180,E1 -25764.293,E2 -25764.293} C_VEL
LIN {X 0,Y 145.456,Z 653.647,A -85,B 0,C 180,E1 -25768.893,E2 -25768.893} C_VEL
LIN {X 0,Y 158.423,Z 648.637,A -85,B 0,C 180,E1 -25773.679,E2 -25773.679} C_VEL
LIN {X 0,Y 163.129,Z 646.612,A -85,B 0,C 180,E1 -25775.058,E2 -25775.058} C_VEL
LIN {X 0,Y 155.661,Z 658.275,A -85,B 0,C 180,E1 -25777.803,E2 -25777.803} C_VEL
LIN {X 0,Y 148.556,Z 668.085,A -85,B 0,C 180,E1 -25780.804,E2 -25780.804} C_VEL
LIN {X 0,Y 141.168,Z 677.419,A -85,B 0,C 180,E1 -25784.598,E2 -25784.598} C_VEL
LIN {X 0,Y 134.967,Z 684.616,A -85,B 0,C 180,E1 -25788.4,E2 -25788.4} C_VEL
LIN {X 0,Y 128.634,Z 691.377,A -85,B 0,C 180,E1 -25793.059,E2 -25793.059} C_VEL
LIN {X 0,Y 122.588,Z 697.637,A -85,B 0,C 180,E1 -25798.937,E2 -25798.937} C_VEL
LIN {X 0,Y 117.886,Z 702.48,A -85,B 0,C 180,E1 -25805.334,E2 -25805.334} C_VEL
LIN {X 0,Y 114.514,Z 706.032,A -85,B 0,C 180,E1 -25812.129,E2 -25812.129} C_VEL
LIN {X 0,Y 112.683,Z 708.374,A -85,B 0,C 180,E1 -25819.215,E2 -25819.215} C_VEL
LIN {X 0,Y 112.059,Z 709.559,A -85,B 0,C 180,E1 -25826.404,E2 -25826.404} C_VEL
LIN {X 0,Y 112.134,Z 709.716,A -85,B 0,C 180,E1 -25830,E2 -25830} C_VEL
LIN {X 0,Y 112.23,Z 709.135,A -85,B 0,C 180,E1 -25837.194,E2 -25837.194} C_VEL
LIN {X 0,Y 113.424,Z 707.412,A -85,B 0,C 180,E1 -25844.35,E2 -25844.35} C_VEL
LIN {X 0,Y 116.019,Z 704.516,A -85,B 0,C 180,E1 -25851.312,E2 -25851.312} C_VEL
LIN {X 0,Y 119.986,Z 700.376,A -85,B 0,C 180,E1 -25857.942,E2 -25857.942} C_VEL
LIN {X 0,Y 125.391,Z 694.883,A -85,B 0,C 180,E1 -25864.089,E2 -25864.089} C_VEL
LIN {X 0,Y 132.01,Z 687.887,A -85,B 0,C 180,E1 -25869.707,E2 -25869.707} C_VEL
LIN {X 0,Y 138.872,Z 680.395,A -85,B 0,C 180,E1 -25874.095,E2 -25874.095} C_VEL
LIN {X 0,Y 145.086,Z 672.743,A -85,B 0,C 180,E1 -25877.621,E2 -25877.621} C_VEL
LIN {X 0,Y 151.986,Z 663.755,A -85,B 0,C 180,E1 -25880.763,E2 -25880.763} C_VEL
LIN {X 0,Y 159.235,Z 653.156,A -85,B 0,C 180,E1 -25883.656,E2 -25883.656} C_VEL
LIN {X 0,Y 166.307,Z 641.599,A -85,B 0,C 180,E1 -25886.03,E2 -25886.03} C_VEL
LIN {X 0,Y 172.819,Z 629.013,A -85,B 0,C 180,E1 -25888.084,E2 -25888.084} C_VEL
LIN {X 0,Y 178.899,Z 615.112,A -85,B 0,C 180,E1 -25889.798,E2 -25889.798} C_VEL
LIN {X 0,Y 184.092,Z 600.603,A -85,B 0,C 180,E1 -25891.125,E2 -25891.125} C_VEL
LIN {X 0,Y 188.355,Z 585.41,A -85,B 0,C 180,E1 -25892.108,E2 -25892.108} C_VEL
LIN {X 0,Y 191.463,Z 569.801,A -85,B 0,C 180,E1 -25892.816,E2 -25892.816} C_VEL
LIN {X 0,Y 193.505,Z 552.475,A -85,B 0,C 180,E1 -25893.348,E2 -25893.348} C_VEL
LIN {X 0,Y 198.611,Z 497.616,A -85,B 0,C 180,E1 -25894.782,E2 -25894.782} C_VEL
LIN {X 0,Y 195.754,Z 489.854,A -85,B 0,C 180,E1 -25897.315,E2 -25897.315} C_VEL
LIN {X 0,Y 193.109,Z 483.563,A -85,B 0,C 180,E1 -25899.911,E2 -25899.911} C_VEL
LIN {X 0,Y 190.131,Z 476.796,A -85,B 0,C 180,E1 -25903.353,E2 -25903.353} C_VEL
